LIN {X 0,Y 527.315,Z 646.786,A -85,B 0,C 180,E1 -4788.874,E2 -4788.874} C_VEL
LIN {X 0,Y 527.547,Z 631.692,A -85,B 0,C 180,E1 -4789.158,E2 -4789.158} C_VEL
LIN {X 0,Y 528.504,Z 486.386,A -85,B 0,C 180,E1 -4791.172,E2 -4791.172} C_VEL
LIN {X 0,Y 526.145,Z 470.012,A -85,B 0,C 180,E1 -4791.511,E2 -4791.511} C_VEL
LIN {X 0,Y 526.763,Z 440.59,A -85,B 0,C 180,E1 -4794.43,E2 -4794.43} C_VEL
LIN {X 0,Y 527.41,Z 413.587,A -85,B 0,C 180,E1 -4797.154,E2 -4797.154} C_VEL
LIN {X 0,Y 528.139,Z 384.774,A -85,B 0,C 180,E1 -4800.122,E2 -4800.122} C_VEL
LIN {X 0,Y 528.004,Z 381.4,A -85,B 0,C 180,E1 -4800.486,E2 -4800.486} C_VEL
LIN {X 0,Y 523.912,Z 365.853,A -85,B 0,C 180,E1 -4802.386,E2 -4802.386} C_VEL
LIN {X 0,Y 523.899,Z 365.848,A -85,B 0,C 180,E1 -4805.227,E2 -4805.227} C_VEL
LIN {X 0,Y 523.892,Z 365.854,A -85,B 0,C 180,E1 -4808.102,E2 -4808.102} C_VEL
LIN {X 0,Y 523.911,Z 365.845,A -85,B 0,C 180,E1 -4811.305,E2 -4811.305} C_VEL
LIN {X 0,Y 523.921,Z 365.841,A -85,B 0,C 180,E1 -4814.688,E2 -4814.688} C_VEL
LIN {X 0,Y 523.877,Z 365.853,A -85,B 0,C 180,E1 -4817.874,E2 -4817.874} C_VEL
LIN {X 0,Y 523.897,Z 365.845,A -85,B 0,C 180,E1 -4820.913,E2 -4820.913} C_VEL
LIN {X 0,Y 523.844,Z 365.856,A -85,B 0,C 180,E1 -4823.821,E2 -4823.821} C_VEL
LIN {X 0,Y 523.896,Z 365.851,A -85,B 0,C 180,E1 -4826.632,E2 -4826.632} C_VEL
LIN {X 0,Y 523.924,Z 365.842,A -85,B 0,C 180,E1 -4829.354,E2 -4829.354} C_VEL
LIN {X 0,Y 523.896,Z 365.854,A -85,B 0,C 180,E1 -4832.295,E2 -4832.295} C_VEL
LIN {X 0,Y 523.887,Z 365.847,A -85,B 0,C 180,E1 -4835.426,E2 -4835.426} C_VEL
LIN {X 0,Y 523.904,Z 365.85,A -85,B 0,C 180,E1 -4837.938,E2 -4837.938} C_VEL
LIN {X 0,Y 523.91,Z 365.854,A -85,B 0,C 180,E1 -4840.406,E2 -4840.406} C_VEL
LIN {X 0,Y 523.903,Z 365.849,A -85,B 0,C 180,E1 -4842.835,E2 -4842.835} C_VEL
LIN {X 0,Y 523.943,Z 365.841,A -85,B 0,C 180,E1 -4845.235,E2 -4845.235} C_VEL
LIN {X 0,Y 523.998,Z 365.842,A -85,B 0,C 180,E1 -4848.394,E2 -4848.394} C_VEL
LIN {X 0,Y 523.937,Z 365.841,A -85,B 0,C 180,E1 -4851.515,E2 -4851.515} C_VEL
LIN {X 0,Y 524.013,Z 365.84,A -85,B 0,C 180,E1 -4854.613,E2 -4854.613} C_VEL
LIN {X 0,Y 524.082,Z 365.82,A -85,B 0,C 180,E1 -4857.695,E2 -4857.695} C_VEL
LIN {X 0,Y 524.104,Z 365.825,A -85,B 0,C 180,E1 -4860.769,E2 -4860.769} C_VEL
LIN {X 0,Y 524.011,Z 365.835,A -85,B 0,C 180,E1 -4863.075,E2 -4863.075} C_VEL
LIN {X 0,Y 523.997,Z 365.832,A -85,B 0,C 180,E1 -4866.16,E2 -4866.16} C_VEL
LIN {X 0,Y 523.962,Z 365.839,A -85,B 0,C 180,E1 -4869.263,E2 -4869.263} C_VEL
LIN {X 0,Y 523.982,Z 365.835,A -85,B 0,C 180,E1 -4871.736,E2 -4871.736} C_VEL
LIN {X 0,Y 523.972,Z 365.838,A -85,B 0,C 180,E1 -4875.05,E2 -4875.05} C_VEL
LIN {X 0,Y 523.933,Z 365.842,A -85,B 0,C 180,E1 -4877.97,E2 -4877.97} C_VEL
LIN {X 0,Y 523.958,Z 365.839,A -85,B 0,C 180,E1 -4880.411,E2 -4880.411} C_VEL
LIN {X 0,Y 523.894,Z 365.854,A -85,B 0,C 180,E1 -4882.895,E2 -4882.895} C_VEL
LIN {X 0,Y 523.884,Z 365.846,A -85,B 0,C 180,E1 -4885.423,E2 -4885.423} C_VEL
LIN {X 0,Y 523.899,Z 365.844,A -85,B 0,C 180,E1 -4888.003,E2 -4888.003} C_VEL
LIN {X 0,Y 523.924,Z 365.849,A -85,B 0,C 180,E1 -4890.854,E2 -4890.854} C_VEL
LIN {X 0,Y 523.919,Z 365.845,A -85,B 0,C 180,E1 -4893.731,E2 -4893.731} C_VEL
LIN {X 0,Y 523.893,Z 365.848,A -85,B 0,C 180,E1 -4896.402,E2 -4896.402} C_VEL
LIN {X 0,Y 523.903,Z 365.852,A -85,B 0,C 180,E1 -4899.087,E2 -4899.087} C_VEL
LIN {X 0,Y 523.9,Z 365.847,A -85,B 0,C 180,E1 -4902.124,E2 -4902.124} C_VEL
LIN {X 0,Y 523.933,Z 365.847,A -85,B 0,C 180,E1 -4905.312,E2 -4905.312} C_VEL
LIN {X 0,Y 523.887,Z 365.852,A -85,B 0,C 180,E1 -4906.926,E2 -4906.926} C_VEL
LIN {X 0,Y 523.209,Z 365.936,A -85,B 0,C 180,E1 -4907.568,E2 -4907.568} C_VEL
LIN {X 0,Y 520.357,Z 366.291,A -85,B 0,C 180,E1 -4908.61,E2 -4908.61} C_VEL
LIN {X 0,Y 517.958,Z 366.589,A -85,B 0,C 180,E1 -4909.449,E2 -4909.449} C_VEL
LIN {X 0,Y 516.933,Z 366.714,A -85,B 0,C 180,E1 -4910.097,E2 -4910.097} C_VEL
LIN {X 0,Y 516.852,Z 366.724,A -85,B 0,C 180,E1 -4910.316,E2 -4910.316} C_VEL
LIN {X 0,Y 516.848,Z 366.729,A -85,B 0,C 180,E1 -4913.348,E2 -4913.348} C_VEL
LIN {X 0,Y 516.876,Z 366.723,A -85,B 0,C 180,E1 -4916.12,E2 -4916.12} C_VEL
LIN {X 0,Y 516.911,Z 366.722,A -85,B 0,C 180,E1 -4919.347,E2 -4919.347} C_VEL
LIN {X 0,Y 516.921,Z 366.886,A -85,B 0,C 180,E1 -4919.682,E2 -4919.682} C_VEL
LIN {X 0,Y 518.76,Z 371.686,A -85,B 0,C 180,E1 -4919.836,E2 -4919.836} C_VEL
LIN {X 0,Y 521.881,Z 378.811,A -85,B 0,C 180,E1 -4920.08,E2 -4920.08} C_VEL
LIN {X 0,Y 521.104,Z 494.688,A -85,B 0,C 180,E1 -4921.74,E2 -4921.74} C_VEL
LIN {X 0,Y 520.916,Z 509.79,A -85,B 0,C 180,E1 -4922.097,E2 -4922.097} C_VEL
LIN {X 0,Y 520.575,Z 523.648,A -85,B 0,C 180,E1 -4922.569,E2 -4922.569} C_VEL
LIN {X 0,Y 520.239,Z 537.825,A -85,B 0,C 180,E1 -4923.213,E2 -4923.213} C_VEL
LIN {X 0,Y 519.763,Z 550.474,A -85,B 0,C 180,E1 -4923.932,E2 -4923.932} C_VEL
LIN {X 0,Y 519.338,Z 562.529,A -85,B 0,C 180,E1 -4924.77,E2 -4924.77} C_VEL
LIN {X 0,Y 518.776,Z 574.916,A -85,B 0,C 180,E1 -4925.808,E2 -4925.808} C_VEL
LIN {X 0,Y 518.289,Z 586.545,A -85,B 0,C 180,E1 -4926.989,E2 -4926.989} C_VEL
LIN {X 0,Y 517.748,Z 597.248,A -85,B 0,C 180,E1 -4928.292,E2 -4928.292} C_VEL
LIN {X 0,Y 517.432,Z 606.116,A -85,B 0,C 180,E1 -4929.586,E2 -4929.586} C_VEL
LIN {X 0,Y 517.053,Z 614.012,A -85,B 0,C 180,E1 -4930.961,E2 -4930.961} C_VEL
LIN {X 0,Y 516.856,Z 620.282,A -85,B 0,C 180,E1 -4932.284,E2 -4932.284} C_VEL
LIN {X 0,Y 516.62,Z 626.219,A -85,B 0,C 180,E1 -4933.807,E2 -4933.807} C_VEL
LIN {X 0,Y 516.515,Z 631.091,A -85,B 0,C 180,E1 -4935.421,E2 -4935.421} C_VEL
LIN {X 0,Y 516.398,Z 633.9,A -85,B 0,C 180,E1 -4936.623,E2 -4936.623} C_VEL
LIN {X 0,Y 516.377,Z 636.848,A -85,B 0,C 180,E1 -4938.504,E2 -4938.504} C_VEL
LIN {X 0,Y 516.313,Z 637.923,A -85,B 0,C 180,E1 -4939.808,E2 -4939.808} C_VEL
LIN {X 0,Y 516.336,Z 638.23,A -85,B 0,C 180,E1 -4941.39,E2 -4941.39} C_VEL
LIN {X 0,Y 516.401,Z 637.436,A -85,B 0,C 180,E1 -4942.965,E2 -4942.965} C_VEL
LIN {X 0,Y 516.42,Z 635.551,A -85,B 0,C 180,E1 -4944.534,E2 -4944.534} C_VEL
LIN {X 0,Y 516.458,Z 632.481,A -85,B 0,C 180,E1 -4946.099,E2 -4946.099} C_VEL
LIN {X 0,Y 516.538,Z 628.218,A -85,B 0,C 180,E1 -4947.661,E2 -4947.661} C_VEL
LIN {X 0,Y 516.697,Z 622.669,A -85,B 0,C 180,E1 -4949.221,E2 -4949.221} C_VEL
LIN {X 0,Y 517.013,Z 615.669,A -85,B 0,C 180,E1 -4950.779,E2 -4950.779} C_VEL
LIN {X 0,Y 517.298,Z 608.205,A -85,B 0,C 180,E1 -4952.141,E2 -4952.141} C_VEL
LIN {X 0,Y 517.678,Z 599.262,A -85,B 0,C 180,E1 -4953.503,E2 -4953.503} C_VEL
LIN {X 0,Y 518.198,Z 588.478,A -85,B 0,C 180,E1 -4954.863,E2 -4954.863} C_VEL
LIN {X 0,Y 518.651,Z 577.402,A -85,B 0,C 180,E1 -4956.028,E2 -4956.028} C_VEL
LIN {X 0,Y 519.169,Z 565.212,A -85,B 0,C 180,E1 -4957.096,E2 -4957.096} C_VEL
LIN {X 0,Y 519.659,Z 553.226,A -85,B 0,C 180,E1 -4957.968,E2 -4957.968} C_VEL
LIN {X 0,Y 520.137,Z 539.655,A -85,B 0,C 180,E1 -4958.775,E2 -4958.775} C_VEL
LIN {X 0,Y 520.55,Z 526.025,A -85,B 0,C 180,E1 -4959.418,E2 -4959.418} C_VEL
LIN {X 0,Y 520.835,Z 510.868,A -85,B 0,C 180,E1 -4959.958,E2 -4959.958} C_VEL
LIN {X 0,Y 521.031,Z 496.258,A -85,B 0,C 180,E1 -4960.32,E2 -4960.32} C_VEL
LIN {X 0,Y 521.839,Z 378.575,A -85,B 0,C 180,E1 -4962.012,E2 -4962.012} C_VEL
LIN {X 0,Y 517.046,Z 367.428,A -85,B 0,C 180,E1 -4962.39,E2 -4962.39} C_VEL
LIN {X 0,Y 516.912,Z 366.723,A -85,B 0,C 180,E1 -4962.424,E2 -4962.424} C_VEL
LIN {X 0,Y 516.833,Z 366.728,A -85,B 0,C 180,E1 -4965.781,E2 -4965.781} C_VEL
LIN {X 0,Y 516.872,Z 366.722,A -85,B 0,C 180,E1 -4968.224,E2 -4968.224} C_VEL
LIN {X 0,Y 516.879,Z 366.726,A -85,B 0,C 180,E1 -4970.703,E2 -4970.703} C_VEL
LIN {X 0,Y 516.836,Z 366.733,A -85,B 0,C 180,E1 -4973.225,E2 -4973.225} C_VEL
LIN {X 0,Y 516.858,Z 366.724,A -85,B 0,C 180,E1 -4976.176,E2 -4976.176} C_VEL
LIN {X 0,Y 516.828,Z 366.729,A -85,B 0,C 180,E1 -4978.42,E2 -4978.42} C_VEL
LIN {X 0,Y 516.847,Z 366.729,A -85,B 0,C 180,E1 -4981.112,E2 -4981.112} C_VEL
LIN {X 0,Y 516.867,Z 366.721,A -85,B 0,C 180,E1 -4983.959,E2 -4983.959} C_VEL
LIN {X 0,Y 516.806,Z 366.733,A -85,B 0,C 180,E1 -4986.751,E2 -4986.751} C_VEL
LIN {X 0,Y 516.841,Z 366.725,A -85,B 0,C 180,E1 -4989.724,E2 -4989.724} C_VEL
LIN {X 0,Y 516.833,Z 366.73,A -85,B 0,C 180,E1 -4992.836,E2 -4992.836} C_VEL
LIN {X 0,Y 516.892,Z 366.724,A -85,B 0,C 180,E1 -4995.006,E2 -4995.006} C_VEL
LIN {X 0,Y 516.844,Z 366.724,A -85,B 0,C 180,E1 -4998.406,E2 -4998.406} C_VEL
LIN {X 0,Y 516.855,Z 366.73,A -85,B 0,C 180,E1 -5001.281,E2 -5001.281} C_VEL
LIN {X 0,Y 516.846,Z 366.725,A -85,B 0,C 180,E1 -5004.217,E2 -5004.217} C_VEL
LIN {X 0,Y 516.852,Z 366.727,A -85,B 0,C 180,E1 -5007.05,E2 -5007.05} C_VEL
LIN {X 0,Y 516.83,Z 366.728,A -85,B 0,C 180,E1 -5009.792,E2 -5009.792} C_VEL
LIN {X 0,Y 516.858,Z 366.723,A -85,B 0,C 180,E1 -5012.463,E2 -5012.463} C_VEL
LIN {X 0,Y 516.847,Z 366.727,A -85,B 0,C 180,E1 -5015.649,E2 -5015.649} C_VEL
LIN {X 0,Y 516.874,Z 366.721,A -85,B 0,C 180,E1 -5018.461,E2 -5018.461} C_VEL
LIN {X 0,Y 516.873,Z 366.722,A -85,B 0,C 180,E1 -5020.953,E2 -5020.953} C_VEL
LIN {X 0,Y 516.874,Z 366.73,A -85,B 0,C 180,E1 -5023.409,E2 -5023.409} C_VEL
LIN {X 0,Y 516.863,Z 366.722,A -85,B 0,C 180,E1 -5025.832,E2 -5025.832} C_VEL
LIN {X 0,Y 516.929,Z 366.705,A -85,B 0,C 180,E1 -5029.027,E2 -5029.027} C_VEL
LIN {X 0,Y 516.91,Z 366.714,A -85,B 0,C 180,E1 -5032.186,E2 -5032.186} C_VEL
LIN {X 0,Y 516.973,Z 366.708,A -85,B 0,C 180,E1 -5034.539,E2 -5034.539} C_VEL
LIN {X 0,Y 517.056,Z 366.701,A -85,B 0,C 180,E1 -5037.663,E2 -5037.663} C_VEL
LIN {X 0,Y 517.045,Z 366.702,A -85,B 0,C 180,E1 -5040,E2 -5040} C_VEL
LIN {X 0,Y 517.058,Z 366.697,A -85,B 0,C 180,E1 -5042.337,E2 -5042.337} C_VEL
LIN {X 0,Y 516.965,Z 366.714,A -85,B 0,C 180,E1 -5045.461,E2 -5045.461} C_VEL
LIN {X 0,Y 516.911,Z 366.714,A -85,B 0,C 180,E1 -5048.601,E2 -5048.601} C_VEL
LIN {X 0,Y 516.942,Z 366.719,A -85,B 0,C 180,E1 -5051.807,E2 -5051.807} C_VEL
LIN {X 0,Y 516.924,Z 366.714,A -85,B 0,C 180,E1 -5055.142,E2 -5055.142} C_VEL
LIN {X 0,Y 516.858,Z 366.723,A -85,B 0,C 180,E1 -5058.224,E2 -5058.224} C_VEL
LIN {X 0,Y 516.86,Z 366.723,A -85,B 0,C 180,E1 -5060.703,E2 -5060.703} C_VEL
LIN {X 0,Y 516.831,Z 366.727,A -85,B 0,C 180,E1 -5063.225,E2 -5063.225} C_VEL
LIN {X 0,Y 516.869,Z 366.723,A -85,B 0,C 180,E1 -5066.182,E2 -5066.182} C_VEL
LIN {X 0,Y 516.875,Z 366.727,A -85,B 0,C 180,E1 -5069.519,E2 -5069.519} C_VEL
LIN {X 0,Y 516.858,Z 366.722,A -85,B 0,C 180,E1 -5072.538,E2 -5072.538} C_VEL
LIN {X 0,Y 516.841,Z 366.727,A -85,B 0,C 180,E1 -5075.327,E2 -5075.327} C_VEL
LIN {X 0,Y 516.854,Z 366.72,A -85,B 0,C 180,E1 -5078.718,E2 -5078.718} C_VEL
LIN {X 0,Y 516.835,Z 366.732,A -85,B 0,C 180,E1 -5081.783,E2 -5081.783} C_VEL
LIN {X 0,Y 516.89,Z 366.719,A -85,B 0,C 180,E1 -5085.007,E2 -5085.007} C_VEL
LIN {X 0,Y 516.829,Z 366.726,A -85,B 0,C 180,E1 -5088.218,E2 -5088.218} C_VEL
LIN {X 0,Y 516.863,Z 366.725,A -85,B 0,C 180,E1 -5091.283,E2 -5091.283} C_VEL
LIN {X 0,Y 516.845,Z 366.728,A -85,B 0,C 180,E1 -5094.674,E2 -5094.674} C_VEL
LIN {X 0,Y 516.918,Z 366.823,A -85,B 0,C 180,E1 -5097.351,E2 -5097.351} C_VEL
LIN {X 0,Y 521.433,Z 384.33,A -85,B 0,C 180,E1 -5099.474,E2 -5099.474} C_VEL
LIN {X 0,Y 520.757,Z 408.762,A -85,B 0,C 180,E1 -5102.033,E2 -5102.033} C_VEL
LIN {X 0,Y 520.055,Z 436.422,A -85,B 0,C 180,E1 -5104.882,E2 -5104.882} C_VEL
LIN {X 0,Y 519.34,Z 465.735,A -85,B 0,C 180,E1 -5107.849,E2 -5107.849} C_VEL
LIN {X 0,Y 519.219,Z 469.127,A -85,B 0,C 180,E1 -5108.189,E2 -5108.189} C_VEL
LIN {X 0,Y 521.848,Z 486.32,A -85,B 0,C 180,E1 -5108.556,E2 -5108.556} C_VEL
LIN {X 0,Y 520.76,Z 638.646,A -85,B 0,C 180,E1 -5110.718,E2 -5110.718} C_VEL
LIN {X 0,Y 520.393,Z 654.328,A -85,B 0,C 180,E1 -5111.102,E2 -5111.102} C_VEL
LIN {X 0,Y 519.991,Z 669.425,A -85,B 0,C 180,E1 -5111.634,E2 -5111.634} C_VEL
LIN {X 0,Y 519.522,Z 683.387,A -85,B 0,C 180,E1 -5112.28,E2 -5112.28} C_VEL
LIN {X 0,Y 519.026,Z 697.119,A -85,B 0,C 180,E1 -5113.075,E2 -5113.075} C_VEL
LIN {X 0,Y 518.522,Z 711.14,A -85,B 0,C 180,E1 -5114.07,E2 -5114.07} C_VEL
LIN {X 0,Y 517.987,Z 723.857,A -85,B 0,C 180,E1 -5115.162,E2 -5115.162} C_VEL
LIN {X 0,Y 517.538,Z 736.378,A -85,B 0,C 180,E1 -5116.453,E2 -5116.453} C_VEL
LIN {X 0,Y 517.111,Z 747.534,A -85,B 0,C 180,E1 -5117.839,E2 -5117.839} C_VEL
LIN {X 0,Y 516.895,Z 756.856,A -85,B 0,C 180,E1 -5119.225,E2 -5119.225} C_VEL
LIN {X 0,Y 516.611,Z 764.583,A -85,B 0,C 180,E1 -5120.604,E2 -5120.604} C_VEL
LIN {X 0,Y 516.508,Z 770.059,A -85,B 0,C 180,E1 -5121.786,E2 -5121.786} C_VEL
LIN {X 0,Y 516.391,Z 774.605,A -85,B 0,C 180,E1 -5122.964,E2 -5122.964} C_VEL
LIN {X 0,Y 516.373,Z 779.385,A -85,B 0,C 180,E1 -5124.533,E2 -5124.533} C_VEL
LIN {X 0,Y 516.307,Z 782.886,A -85,B 0,C 180,E1 -5126.097,E2 -5126.097} C_VEL
LIN {X 0,Y 516.257,Z 785.188,A -85,B 0,C 180,E1 -5127.659,E2 -5127.659} C_VEL
LIN {X 0,Y 516.157,Z 786.347,A -85,B 0,C 180,E1 -5129.22,E2 -5129.22} C_VEL
LIN {X 0,Y 516.157,Z 786.346,A -85,B 0,C 180,E1 -5130.78,E2 -5130.78} C_VEL
LIN {X 0,Y 516.257,Z 785.185,A -85,B 0,C 180,E1 -5132.34,E2 -5132.34} C_VEL
LIN {X 0,Y 516.307,Z 782.882,A -85,B 0,C 180,E1 -5133.902,E2 -5133.902} C_VEL
LIN {X 0,Y 516.372,Z 779.387,A -85,B 0,C 180,E1 -5135.467,E2 -5135.467} C_VEL
LIN {X 0,Y 516.391,Z 774.611,A -85,B 0,C 180,E1 -5137.035,E2 -5137.035} C_VEL
LIN {X 0,Y 516.54,Z 768.361,A -85,B 0,C 180,E1 -5138.607,E2 -5138.607} C_VEL
LIN {X 0,Y 516.676,Z 761.44,A -85,B 0,C 180,E1 -5139.987,E2 -5139.987} C_VEL
LIN {X 0,Y 516.952,Z 753.027,A -85,B 0,C 180,E1 -5141.368,E2 -5141.368} C_VEL
LIN {X 0,Y 517.283,Z 742.958,A -85,B 0,C 180,E1 -5142.754,E2 -5142.754} C_VEL
LIN {X 0,Y 517.649,Z 732.687,A -85,B 0,C 180,E1 -5143.944,E2 -5143.944} C_VEL
LIN {X 0,Y 518.079,Z 720.663,A -85,B 0,C 180,E1 -5145.124,E2 -5145.124} C_VEL
LIN {X 0,Y 518.59,Z 708.438,A -85,B 0,C 180,E1 -5146.129,E2 -5146.129} C_VEL
LIN {X 0,Y 519.071,Z 695.419,A -85,B 0,C 180,E1 -5147.024,E2 -5147.024} C_VEL
LIN {X 0,Y 519.566,Z 681.262,A -85,B 0,C 180,E1 -5147.82,E2 -5147.82} C_VEL
LIN {X 0,Y 520.026,Z 666.743,A -85,B 0,C 180,E1 -5148.466,E2 -5148.466} C_VEL
LIN {X 0,Y 520.439,Z 651.075,A -85,B 0,C 180,E1 -5148.986,E2 -5148.986} C_VEL
LIN {X 0,Y 520.798,Z 636.224,A -85,B 0,C 180,E1 -5149.321,E2 -5149.321} C_VEL
LIN {X 0,Y 521.835,Z 486.88,A -85,B 0,C 180,E1 -5151.433,E2 -5151.433} C_VEL
LIN {X 0,Y 519.194,Z 468.922,A -85,B 0,C 180,E1 -5151.812,E2 -5151.812} C_VEL
LIN {X 0,Y 519.864,Z 440.568,A -85,B 0,C 180,E1 -5154.669,E2 -5154.669} C_VEL
LIN {X 0,Y 520.564,Z 414.648,A -85,B 0,C 180,E1 -5157.323,E2 -5157.323} C_VEL
LIN {X 0,Y 521.371,Z 386.766,A -85,B 0,C 180,E1 -5160.24,E2 -5160.24} C_VEL
LIN {X 0,Y 521.416,Z 384.129,A -85,B 0,C 180,E1 -5160.522,E2 -5160.522} C_VEL
LIN {X 0,Y 516.889,Z 366.725,A -85,B 0,C 180,E1 -5162.708,E2 -5162.708} C_VEL
LIN {X 0,Y 516.807,Z 366.734,A -85,B 0,C 180,E1 -5165.784,E2 -5165.784} C_VEL
LIN {X 0,Y 516.864,Z 366.726,A -85,B 0,C 180,E1 -5168.716,E2 -5168.716} C_VEL
LIN {X 0,Y 516.872,Z 366.725,A -85,B 0,C 180,E1 -5171.777,E2 -5171.777} C_VEL
LIN {X 0,Y 516.886,Z 366.715,A -85,B 0,C 180,E1 -5175.006,E2 -5175.006} C_VEL
LIN {X 0,Y 516.838,Z 366.73,A -85,B 0,C 180,E1 -5178.406,E2 -5178.406} C_VEL
LIN {X 0,Y 516.859,Z 366.721,A -85,B 0,C 180,E1 -5181.282,E2 -5181.282} C_VEL
LIN {X 0,Y 516.837,Z 366.73,A -85,B 0,C 180,E1 -5184.672,E2 -5184.672} C_VEL
LIN {X 0,Y 516.854,Z 366.724,A -85,B 0,C 180,E1 -5187.461,E2 -5187.461} C_VEL
LIN {X 0,Y 516.871,Z 366.73,A -85,B 0,C 180,E1 -5190.481,E2 -5190.481} C_VEL
LIN {X 0,Y 516.864,Z 366.725,A -85,B 0,C 180,E1 -5193.818,E2 -5193.818} C_VEL
LIN {X 0,Y 516.826,Z 366.732,A -85,B 0,C 180,E1 -5196.775,E2 -5196.775} C_VEL
LIN {X 0,Y 516.86,Z 366.723,A -85,B 0,C 180,E1 -5199.751,E2 -5199.751} C_VEL
LIN {X 0,Y 516.862,Z 366.729,A -85,B 0,C 180,E1 -5202.594,E2 -5202.594} C_VEL
LIN {X 0,Y 516.914,Z 366.718,A -85,B 0,C 180,E1 -5205.029,E2 -5205.029} C_VEL
LIN {X 0,Y 516.951,Z 366.718,A -85,B 0,C 180,E1 -5208.234,E2 -5208.234} C_VEL
LIN {X 0,Y 516.909,Z 366.717,A -85,B 0,C 180,E1 -5211.399,E2 -5211.399} C_VEL
LIN {X 0,Y 516.963,Z 366.717,A -85,B 0,C 180,E1 -5214.539,E2 -5214.539} C_VEL
LIN {X 0,Y 517.054,Z 366.696,A -85,B 0,C 180,E1 -5217.663,E2 -5217.663} C_VEL
LIN {X 0,Y 517.074,Z 366.7,A -85,B 0,C 180,E1 -5220.779,E2 -5220.779} C_VEL
LIN {X 0,Y 516.953,Z 366.714,A -85,B 0,C 180,E1 -5223.118,E2 -5223.118} C_VEL
LIN {X 0,Y 516.966,Z 366.708,A -85,B 0,C 180,E1 -5226.244,E2 -5226.244} C_VEL
LIN {X 0,Y 516.918,Z 366.715,A -85,B 0,C 180,E1 -5229.39,E2 -5229.39} C_VEL
LIN {X 0,Y 516.938,Z 366.713,A -85,B 0,C 180,E1 -5231.807,E2 -5231.807} C_VEL
LIN {X 0,Y 516.924,Z 366.714,A -85,B 0,C 180,E1 -5235.144,E2 -5235.144} C_VEL
LIN {X 0,Y 516.901,Z 366.72,A -85,B 0,C 180,E1 -5238.223,E2 -5238.223} C_VEL
LIN {X 0,Y 516.898,Z 366.717,A -85,B 0,C 180,E1 -5240.702,E2 -5240.702} C_VEL
LIN {X 0,Y 516.871,Z 366.723,A -85,B 0,C 180,E1 -5244.074,E2 -5244.074} C_VEL
LIN {X 0,Y 516.827,Z 366.728,A -85,B 0,C 180,E1 -5246.664,E2 -5246.664} C_VEL
LIN {X 0,Y 516.895,Z 366.721,A -85,B 0,C 180,E1 -5249.524,E2 -5249.524} C_VEL
LIN {X 0,Y 516.883,Z 366.719,A -85,B 0,C 180,E1 -5252.544,E2 -5252.544} C_VEL
LIN {X 0,Y 516.855,Z 366.726,A -85,B 0,C 180,E1 -5255.33,E2 -5255.33} C_VEL
LIN {X 0,Y 516.869,Z 366.722,A -85,B 0,C 180,E1 -5257.944,E2 -5257.944} C_VEL
LIN {X 0,Y 516.845,Z 366.728,A -85,B 0,C 180,E1 -5260.746,E2 -5260.746} C_VEL
LIN {X 0,Y 516.873,Z 366.718,A -85,B 0,C 180,E1 -5263.905,E2 -5263.905} C_VEL
LIN {X 0,Y 516.837,Z 366.728,A -85,B 0,C 180,E1 -5266.928,E2 -5266.928} C_VEL
LIN {X 0,Y 516.854,Z 366.725,A -85,B 0,C 180,E1 -5269.594,E2 -5269.594} C_VEL
LIN {X 0,Y 516.852,Z 366.724,A -85,B 0,C 180,E1 -5270.316,E2 -5270.316} C_VEL
LIN {X 0,Y 516.193,Z 366.814,A -85,B 0,C 180,E1 -5270.966,E2 -5270.966} C_VEL
LIN {X 0,Y 513.344,Z 367.167,A -85,B 0,C 180,E1 -5272.022,E2 -5272.022} C_VEL
LIN {X 0,Y 510.929,Z 367.467,A -85,B 0,C 180,E1 -5272.873,E2 -5272.873} C_VEL
LIN {X 0,Y 509.887,Z 367.594,A -85,B 0,C 180,E1 -5273.529,E2 -5273.529} C_VEL
LIN {X 0,Y 509.8,Z 367.603,A -85,B 0,C 180,E1 -5273.752,E2 -5273.752} C_VEL
LIN {X 0,Y 509.835,Z 367.603,A -85,B 0,C 180,E1 -5276.539,E2 -5276.539} C_VEL
LIN {X 0,Y 509.877,Z 367.625,A -85,B 0,C 180,E1 -5279.363,E2 -5279.363} C_VEL
LIN {X 0,Y 511.415,Z 371.854,A -85,B 0,C 180,E1 -5279.499,E2 -5279.499} C_VEL
LIN {X 0,Y 515.302,Z 380.765,A -85,B 0,C 180,E1 -5279.812,E2 -5279.812} C_VEL
LIN {X 0,Y 514.445,Z 495.575,A -85,B 0,C 180,E1 -5281.479,E2 -5281.479} C_VEL
LIN {X 0,Y 514.256,Z 510.81,A -85,B 0,C 180,E1 -5281.842,E2 -5281.842} C_VEL
LIN {X 0,Y 513.941,Z 525.052,A -85,B 0,C 180,E1 -5282.337,E2 -5282.337} C_VEL
LIN {X 0,Y 513.586,Z 538.387,A -85,B 0,C 180,E1 -5282.95,E2 -5282.95} C_VEL
LIN {X 0,Y 513.075,Z 551.1,A -85,B 0,C 180,E1 -5283.676,E2 -5283.676} C_VEL
LIN {X 0,Y 512.635,Z 563.228,A -85,B 0,C 180,E1 -5284.525,E2 -5284.525} C_VEL
LIN {X 0,Y 512.015,Z 575.76,A -85,B 0,C 180,E1 -5285.584,E2 -5285.584} C_VEL
LIN {X 0,Y 511.529,Z 586.663,A -85,B 0,C 180,E1 -5286.693,E2 -5286.693} C_VEL
LIN {X 0,Y 510.957,Z 597.337,A -85,B 0,C 180,E1 -5287.988,E2 -5287.988} C_VEL
LIN {X 0,Y 510.57,Z 606.929,A -85,B 0,C 180,E1 -5289.394,E2 -5289.394} C_VEL
LIN {X 0,Y 510.127,Z 615.442,A -85,B 0,C 180,E1 -5290.902,E2 -5290.902} C_VEL
LIN {X 0,Y 509.858,Z 622.115,A -85,B 0,C 180,E1 -5292.348,E2 -5292.348} C_VEL
LIN {X 0,Y 509.648,Z 628.21,A -85,B 0,C 180,E1 -5293.991,E2 -5293.991} C_VEL
LIN {X 0,Y 509.479,Z 632.835,A -85,B 0,C 180,E1 -5295.624,E2 -5295.624} C_VEL
LIN {X 0,Y 509.353,Z 636.146,A -85,B 0,C 180,E1 -5297.247,E2 -5297.247} C_VEL
LIN {X 0,Y 509.362,Z 638.239,A -85,B 0,C 180,E1 -5298.863,E2 -5298.863} C_VEL
LIN {X 0,Y 509.302,Z 639.205,A -85,B 0,C 180,E1 -5300.469,E2 -5300.469} C_VEL
LIN {X 0,Y 509.337,Z 639.056,A -85,B 0,C 180,E1 -5302.069,E2 -5302.069} C_VEL
LIN {X 0,Y 509.416,Z 637.793,A -85,B 0,C 180,E1 -5303.664,E2 -5303.664} C_VEL
LIN {X 0,Y 509.388,Z 635.392,A -85,B 0,C 180,E1 -5305.252,E2 -5305.252} C_VEL
LIN {X 0,Y 509.576,Z 631.807,A -85,B 0,C 180,E1 -5306.838,E2 -5306.838} C_VEL
LIN {X 0,Y 509.593,Z 627.042,A -85,B 0,C 180,E1 -5308.42,E2 -5308.42} C_VEL
LIN {X 0,Y 509.854,Z 620.902,A -85,B 0,C 180,E1 -5310,E2 -5310} C_VEL
LIN {X 0,Y 510.217,Z 613.234,A -85,B 0,C 180,E1 -5311.579,E2 -5311.579} C_VEL
LIN {X 0,Y 510.565,Z 605.095,A -85,B 0,C 180,E1 -5312.959,E2 -5312.959} C_VEL
LIN {X 0,Y 511.094,Z 595.303,A -85,B 0,C 180,E1 -5314.338,E2 -5314.338} C_VEL
LIN {X 0,Y 511.572,Z 585.332,A -85,B 0,C 180,E1 -5315.519,E2 -5315.519} C_VEL
LIN {X 0,Y 512.067,Z 573.425,A -85,B 0,C 180,E1 -5316.7,E2 -5316.7} C_VEL
LIN {X 0,Y 512.638,Z 561.493,A -85,B 0,C 180,E1 -5317.682,E2 -5317.682} C_VEL
LIN {X 0,Y 513.193,Z 548.475,A -85,B 0,C 180,E1 -5318.565,E2 -5318.565} C_VEL
LIN {X 0,Y 513.613,Z 535.982,A -85,B 0,C 180,E1 -5319.252,E2 -5319.252} C_VEL
LIN {X 0,Y 514.013,Z 522.246,A -85,B 0,C 180,E1 -5319.851,E2 -5319.851} C_VEL
LIN {X 0,Y 514.252,Z 507.515,A -85,B 0,C 180,E1 -5320.333,E2 -5320.333} C_VEL
LIN {X 0,Y 514.401,Z 492.958,A -85,B 0,C 180,E1 -5320.654,E2 -5320.654} C_VEL
LIN {X 0,Y 515.255,Z 380.378,A -85,B 0,C 180,E1 -5322.28,E2 -5322.28} C_VEL
LIN {X 0,Y 509.971,Z 368.313,A -85,B 0,C 180,E1 -5322.703,E2 -5322.703} C_VEL
LIN {X 0,Y 509.851,Z 367.604,A -85,B 0,C 180,E1 -5322.741,E2 -5322.741} C_VEL
LIN {X 0,Y 509.801,Z 367.604,A -85,B 0,C 180,E1 -5326.005,E2 -5326.005} C_VEL
LIN {X 0,Y 509.829,Z 367.602,A -85,B 0,C 180,E1 -5328.485,E2 -5328.485} C_VEL
LIN {X 0,Y 509.824,Z 367.608,A -85,B 0,C 180,E1 -5331.003,E2 -5331.003} C_VEL
LIN {X 0,Y 509.797,Z 367.606,A -85,B 0,C 180,E1 -5333.565,E2 -5333.565} C_VEL
LIN {X 0,Y 509.799,Z 367.605,A -85,B 0,C 180,E1 -5336.352,E2 -5336.352} C_VEL
LIN {X 0,Y 509.792,Z 367.611,A -85,B 0,C 180,E1 -5338.849,E2 -5338.849} C_VEL
LIN {X 0,Y 509.786,Z 367.607,A -85,B 0,C 180,E1 -5341.592,E2 -5341.592} C_VEL
LIN {X 0,Y 509.826,Z 367.599,A -85,B 0,C 180,E1 -5344.415,E2 -5344.415} C_VEL
LIN {X 0,Y 509.774,Z 367.612,A -85,B 0,C 180,E1 -5347.344,E2 -5347.344} C_VEL
LIN {X 0,Y 509.79,Z 367.602,A -85,B 0,C 180,E1 -5350.386,E2 -5350.386} C_VEL
LIN {X 0,Y 509.787,Z 367.606,A -85,B 0,C 180,E1 -5353.574,E2 -5353.574} C_VEL
LIN {X 0,Y 509.787,Z 367.604,A -85,B 0,C 180,E1 -5356.424,E2 -5356.424} C_VEL
LIN {X 0,Y 509.807,Z 367.605,A -85,B 0,C 180,E1 -5359.614,E2 -5359.614} C_VEL
LIN {X 0,Y 509.781,Z 367.605,A -85,B 0,C 180,E1 -5362.656,E2 -5362.656} C_VEL
LIN {X 0,Y 509.825,Z 367.598,A -85,B 0,C 180,E1 -5365.801,E2 -5365.801} C_VEL
LIN {X 0,Y 509.807,Z 367.604,A -85,B 0,C 180,E1 -5368.726,E2 -5368.726} C_VEL
LIN {X 0,Y 509.815,Z 367.601,A -85,B 0,C 180,E1 -5372.05,E2 -5372.05} C_VEL
LIN {X 0,Y 509.773,Z 367.607,A -85,B 0,C 180,E1 -5374.698,E2 -5374.698} C_VEL
LIN {X 0,Y 509.816,Z 367.608,A -85,B 0,C 180,E1 -5377.458,E2 -5377.458} C_VEL
LIN {X 0,Y 509.898,Z 367.591,A -85,B 0,C 180,E1 -5379.844,E2 -5379.844} C_VEL
LIN {X 0,Y 509.843,Z 367.601,A -85,B 0,C 180,E1 -5383.173,E2 -5383.173} C_VEL
LIN {X 0,Y 509.836,Z 367.6,A -85,B 0,C 180,E1 -5385.633,E2 -5385.633} C_VEL
LIN {X 0,Y 509.894,Z 367.579,A -85,B 0,C 180,E1 -5388.874,E2 -5388.874} C_VEL
LIN {X 0,Y 509.863,Z 367.593,A -85,B 0,C 180,E1 -5392.077,E2 -5392.077} C_VEL
LIN {X 0,Y 509.928,Z 367.586,A -85,B 0,C 180,E1 -5394.463,E2 -5394.463} C_VEL
LIN {X 0,Y 510.025,Z 367.577,A -85,B 0,C 180,E1 -5397.631,E2 -5397.631} C_VEL
LIN {X 0,Y 510.015,Z 367.578,A -85,B 0,C 180,E1 -5400,E2 -5400} C_VEL
LIN {X 0,Y 510.029,Z 367.572,A -85,B 0,C 180,E1 -5402.369,E2 -5402.369} C_VEL
LIN {X 0,Y 509.918,Z 367.593,A -85,B 0,C 180,E1 -5405.536,E2 -5405.536} C_VEL
LIN {X 0,Y 509.865,Z 367.596,A -85,B 0,C 180,E1 -5407.923,E2 -5407.923} C_VEL
LIN {X 0,Y 509.896,Z 367.592,A -85,B 0,C 180,E1 -5411.126,E2 -5411.126} C_VEL
LIN {X 0,Y 509.83,Z 367.596,A -85,B 0,C 180,E1 -5414.367,E2 -5414.367} C_VEL
LIN {X 0,Y 509.778,Z 367.606,A -85,B 0,C 180,E1 -5416.829,E2 -5416.829} C_VEL
LIN {X 0,Y 509.814,Z 367.602,A -85,B 0,C 180,E1 -5419.32,E2 -5419.32} C_VEL
LIN {X 0,Y 509.814,Z 367.599,A -85,B 0,C 180,E1 -5422.541,E2 -5422.541} C_VEL
LIN {X 0,Y 509.791,Z 367.607,A -85,B 0,C 180,E1 -5425.3,E2 -5425.3} C_VEL
LIN {X 0,Y 509.8,Z 367.606,A -85,B 0,C 180,E1 -5428.082,E2 -5428.082} C_VEL
LIN {X 0,Y 509.819,Z 367.601,A -85,B 0,C 180,E1 -5430.667,E2 -5430.667} C_VEL
LIN {X 0,Y 509.824,Z 367.602,A -85,B 0,C 180,E1 -5433.463,E2 -5433.463} C_VEL
LIN {X 0,Y 509.757,Z 367.611,A -85,B 0,C 180,E1 -5436.359,E2 -5436.359} C_VEL
LIN {X 0,Y 509.802,Z 367.603,A -85,B 0,C 180,E1 -5439.467,E2 -5439.467} C_VEL
LIN {X 0,Y 509.778,Z 367.605,A -85,B 0,C 180,E1 -5442.495,E2 -5442.495} C_VEL
LIN {X 0,Y 509.833,Z 367.6,A -85,B 0,C 180,E1 -5445.33,E2 -5445.33} C_VEL
LIN {X 0,Y 509.78,Z 367.601,A -85,B 0,C 180,E1 -5448.568,E2 -5448.568} C_VEL
LIN {X 0,Y 509.808,Z 367.608,A -85,B 0,C 180,E1 -5451.659,E2 -5451.659} C_VEL
LIN {X 0,Y 509.803,Z 367.606,A -85,B 0,C 180,E1 -5454.62,E2 -5454.62} C_VEL
LIN {X 0,Y 509.858,Z 367.616,A -85,B 0,C 180,E1 -5457.063,E2 -5457.063} C_VEL
LIN {X 0,Y 514.667,Z 386.214,A -85,B 0,C 180,E1 -5459.349,E2 -5459.349} C_VEL
LIN {X 0,Y 513.946,Z 409.84,A -85,B 0,C 180,E1 -5461.851,E2 -5461.851} C_VEL
LIN {X 0,Y 513.192,Z 436.826,A -85,B 0,C 180,E1 -5464.668,E2 -5464.668} C_VEL
LIN {X 0,Y 512.373,Z 466.644,A -85,B 0,C 180,E1 -5467.734,E2 -5467.734} C_VEL
LIN {X 0,Y 512.308,Z 468.297,A -85,B 0,C 180,E1 -5467.892,E2 -5467.892} C_VEL
LIN {X 0,Y 515.198,Z 487.539,A -85,B 0,C 180,E1 -5468.298,E2 -5468.298} C_VEL
LIN {X 0,Y 514.052,Z 636.943,A -85,B 0,C 180,E1 -5470.443,E2 -5470.443} C_VEL
LIN {X 0,Y 513.616,Z 652.848,A -85,B 0,C 180,E1 -5470.828,E2 -5470.828} C_VEL
LIN {X 0,Y 513.169,Z 668.596,A -85,B 0,C 180,E1 -5471.39,E2 -5471.39} C_VEL
LIN {X 0,Y 512.638,Z 682.352,A -85,B 0,C 180,E1 -5472.034,E2 -5472.034} C_VEL
LIN {X 0,Y 512.142,Z 696.091,A -85,B 0,C 180,E1 -5472.84,E2 -5472.84} C_VEL
LIN {X 0,Y 511.608,Z 708.787,A -85,B 0,C 180,E1 -5473.746,E2 -5473.746} C_VEL
LIN {X 0,Y 511.006,Z 721.725,A -85,B 0,C 180,E1 -5474.852,E2 -5474.852} C_VEL
LIN {X 0,Y 510.564,Z 733.526,A -85,B 0,C 180,E1 -5476.061,E2 -5476.061} C_VEL
LIN {X 0,Y 510.191,Z 743.484,A -85,B 0,C 180,E1 -5477.267,E2 -5477.267} C_VEL
LIN {X 0,Y 509.889,Z 753.423,A -85,B 0,C 180,E1 -5478.693,E2 -5478.693} C_VEL
LIN {X 0,Y 509.576,Z 761.468,A -85,B 0,C 180,E1 -5480.073,E2 -5480.073} C_VEL
LIN {X 0,Y 509.431,Z 769.133,A -85,B 0,C 180,E1 -5481.671,E2 -5481.671} C_VEL
LIN {X 0,Y 509.289,Z 775.219,A -85,B 0,C 180,E1 -5483.264,E2 -5483.264} C_VEL
LIN {X 0,Y 509.305,Z 778.85,A -85,B 0,C 180,E1 -5484.457,E2 -5484.457} C_VEL
LIN {X 0,Y 509.217,Z 782.511,A -85,B 0,C 180,E1 -5486.043,E2 -5486.043} C_VEL
LIN {X 0,Y 509.185,Z 784.924,A -85,B 0,C 180,E1 -5487.627,E2 -5487.627} C_VEL
LIN {X 0,Y 509.071,Z 786.123,A -85,B 0,C 180,E1 -5489.209,E2 -5489.209} C_VEL
LIN {X 0,Y 509.071,Z 786.122,A -85,B 0,C 180,E1 -5490.791,E2 -5490.791} C_VEL
LIN {X 0,Y 509.185,Z 784.921,A -85,B 0,C 180,E1 -5492.373,E2 -5492.373} C_VEL
LIN {X 0,Y 509.217,Z 782.506,A -85,B 0,C 180,E1 -5493.957,E2 -5493.957} C_VEL
LIN {X 0,Y 509.303,Z 778.848,A -85,B 0,C 180,E1 -5495.543,E2 -5495.543} C_VEL
LIN {X 0,Y 509.317,Z 773.837,A -85,B 0,C 180,E1 -5497.133,E2 -5497.133} C_VEL
LIN {X 0,Y 509.483,Z 767.373,A -85,B 0,C 180,E1 -5498.727,E2 -5498.727} C_VEL
LIN {X 0,Y 509.687,Z 759.266,A -85,B 0,C 180,E1 -5500.326,E2 -5500.326} C_VEL
LIN {X 0,Y 509.898,Z 750.521,A -85,B 0,C 180,E1 -5501.748,E2 -5501.748} C_VEL
LIN {X 0,Y 510.311,Z 740.321,A -85,B 0,C 180,E1 -5503.134,E2 -5503.134} C_VEL
LIN {X 0,Y 510.691,Z 729.777,A -85,B 0,C 180,E1 -5504.341,E2 -5504.341} C_VEL
LIN {X 0,Y 511.248,Z 716.867,A -85,B 0,C 180,E1 -5505.582,E2 -5505.582} C_VEL
LIN {X 0,Y 511.775,Z 703.337,A -85,B 0,C 180,E1 -5506.658,E2 -5506.658} C_VEL
LIN {X 0,Y 512.388,Z 689.45,A -85,B 0,C 180,E1 -5507.562,E2 -5507.562} C_VEL
LIN {X 0,Y 512.902,Z 675.1,A -85,B 0,C 180,E1 -5508.318,E2 -5508.318} C_VEL
LIN {X 0,Y 513.407,Z 659.511,A -85,B 0,C 180,E1 -5508.95,E2 -5508.95} C_VEL
LIN {X 0,Y 513.848,Z 644.317,A -85,B 0,C 180,E1 -5509.395,E2 -5509.395} C_VEL
LIN {X 0,Y 514.116,Z 628.274,A -85,B 0,C 180,E1 -5509.697,E2 -5509.697} C_VEL
LIN {X 0,Y 515.193,Z 487.821,A -85,B 0,C 180,E1 -5511.695,E2 -5511.695} C_VEL
LIN {X 0,Y 512.269,Z 467.76,A -85,B 0,C 180,E1 -5512.128,E2 -5512.128} C_VEL
LIN {X 0,Y 513.058,Z 438.478,A -85,B 0,C 180,E1 -5515.127,E2 -5515.127} C_VEL
LIN {X 0,Y 513.783,Z 413.651,A -85,B 0,C 180,E1 -5517.715,E2 -5517.715} C_VEL
LIN {X 0,Y 514.662,Z 386.128,A -85,B 0,C 180,E1 -5520.65,E2 -5520.65} C_VEL
LIN {X 0,Y 510.491,Z 370.102,A -85,B 0,C 180,E1 -5522.674,E2 -5522.674} C_VEL
LIN {X 0,Y 509.834,Z 367.603,A -85,B 0,C 180,E1 -5523.03,E2 -5523.03} C_VEL
LIN {X 0,Y 509.787,Z 367.609,A -85,B 0,C 180,E1 -5525.572,E2 -5525.572} C_VEL
LIN {X 0,Y 509.806,Z 367.609,A -85,B 0,C 180,E1 -5528.34,E2 -5528.34} C_VEL
LIN {X 0,Y 509.82,Z 367.601,A -85,B 0,C 180,E1 -5531.427,E2 -5531.427} C_VEL
LIN {X 0,Y 509.829,Z 367.596,A -85,B 0,C 180,E1 -5534.669,E2 -5534.669} C_VEL
LIN {X 0,Y 509.774,Z 367.606,A -85,B 0,C 180,E1 -5537.504,E2 -5537.504} C_VEL
LIN {X 0,Y 509.819,Z 367.601,A -85,B 0,C 180,E1 -5540.645,E2 -5540.645} C_VEL
LIN {X 0,Y 509.753,Z 367.61,A -85,B 0,C 180,E1 -5543.641,E2 -5543.641} C_VEL
LIN {X 0,Y 509.82,Z 367.606,A -85,B 0,C 180,E1 -5546.536,E2 -5546.536} C_VEL
LIN {X 0,Y 509.814,Z 367.6,A -85,B 0,C 180,E1 -5549.332,E2 -5549.332} C_VEL
LIN {X 0,Y 509.809,Z 367.608,A -85,B 0,C 180,E1 -5552.05,E2 -5552.05} C_VEL
LIN {X 0,Y 509.786,Z 367.608,A -85,B 0,C 180,E1 -5554.699,E2 -5554.699} C_VEL
LIN {X 0,Y 509.809,Z 367.603,A -85,B 0,C 180,E1 -5557.459,E2 -5557.459} C_VEL
LIN {X 0,Y 509.809,Z 367.607,A -85,B 0,C 180,E1 -5560.68,E2 -5560.68} C_VEL
LIN {X 0,Y 509.779,Z 367.606,A -85,B 0,C 180,E1 -5563.171,E2 -5563.171} C_VEL
LIN {X 0,Y 509.824,Z 367.599,A -85,B 0,C 180,E1 -5565.633,E2 -5565.633} C_VEL
LIN {X 0,Y 509.89,Z 367.593,A -85,B 0,C 180,E1 -5568.874,E2 -5568.874} C_VEL
LIN {X 0,Y 509.861,Z 367.598,A -85,B 0,C 180,E1 -5572.077,E2 -5572.077} C_VEL
LIN {X 0,Y 509.916,Z 367.593,A -85,B 0,C 180,E1 -5574.464,E2 -5574.464} C_VEL
LIN {X 0,Y 510.025,Z 367.571,A -85,B 0,C 180,E1 -5577.631,E2 -5577.631} C_VEL
LIN {X 0,Y 510.045,Z 367.575,A -85,B 0,C 180,E1 -5580.79,E2 -5580.79} C_VEL
LIN {X 0,Y 509.895,Z 367.592,A -85,B 0,C 180,E1 -5583.161,E2 -5583.161} C_VEL
LIN {X 0,Y 509.92,Z 367.585,A -85,B 0,C 180,E1 -5586.331,E2 -5586.331} C_VEL
LIN {X 0,Y 509.868,Z 367.595,A -85,B 0,C 180,E1 -5588.721,E2 -5588.721} C_VEL
LIN {X 0,Y 509.89,Z 367.591,A -85,B 0,C 180,E1 -5591.932,E2 -5591.932} C_VEL
LIN {X 0,Y 509.881,Z 367.59,A -85,B 0,C 180,E1 -5595.242,E2 -5595.242} C_VEL
LIN {X 0,Y 509.846,Z 367.602,A -85,B 0,C 180,E1 -5598.485,E2 -5598.485} C_VEL
LIN {X 0,Y 509.836,Z 367.596,A -85,B 0,C 180,E1 -5601.003,E2 -5601.003} C_VEL
LIN {X 0,Y 509.805,Z 367.603,A -85,B 0,C 180,E1 -5603.565,E2 -5603.565} C_VEL
LIN {X 0,Y 509.802,Z 367.602,A -85,B 0,C 180,E1 -5606.357,E2 -5606.357} C_VEL
LIN {X 0,Y 509.836,Z 367.605,A -85,B 0,C 180,E1 -5608.847,E2 -5608.847} C_VEL
LIN {X 0,Y 509.806,Z 367.597,A -85,B 0,C 180,E1 -5611.591,E2 -5611.591} C_VEL
LIN {X 0,Y 509.828,Z 367.603,A -85,B 0,C 180,E1 -5614.416,E2 -5614.416} C_VEL
LIN {X 0,Y 509.806,Z 367.605,A -85,B 0,C 180,E1 -5617.342,E2 -5617.342} C_VEL
LIN {X 0,Y 509.805,Z 367.603,A -85,B 0,C 180,E1 -5620.386,E2 -5620.386} C_VEL
LIN {X 0,Y 509.787,Z 367.608,A -85,B 0,C 180,E1 -5623.06,E2 -5623.06} C_VEL
LIN {X 0,Y 509.815,Z 367.602,A -85,B 0,C 180,E1 -5625.795,E2 -5625.795} C_VEL
LIN {X 0,Y 509.826,Z 367.603,A -85,B 0,C 180,E1 -5628.573,E2 -5628.573} C_VEL
LIN {X 0,Y 509.844,Z 367.596,A -85,B 0,C 180,E1 -5631.788,E2 -5631.788} C_VEL
LIN {X 0,Y 509.8,Z 367.603,A -85,B 0,C 180,E1 -5633.752,E2 -5633.752} C_VEL
LIN {X 0,Y 509.136,Z 367.686,A -85,B 0,C 180,E1 -5634.412,E2 -5634.412} C_VEL
LIN {X 0,Y 506.311,Z 368.043,A -85,B 0,C 180,E1 -5635.483,E2 -5635.483} C_VEL
LIN {X 0,Y 503.915,Z 368.344,A -85,B 0,C 180,E1 -5636.347,E2 -5636.347} C_VEL
LIN {X 0,Y 502.873,Z 368.473,A -85,B 0,C 180,E1 -5637.013,E2 -5637.013} C_VEL
LIN {X 0,Y 502.78,Z 368.481,A -85,B 0,C 180,E1 -5637.239,E2 -5637.239} C_VEL
LIN {X 0,Y 502.824,Z 368.475,A -85,B 0,C 180,E1 -5639.016,E2 -5639.016} C_VEL
LIN {X 0,Y 503.897,Z 371.449,A -85,B 0,C 180,E1 -5639.13,E2 -5639.13} C_VEL
LIN {X 0,Y 508.668,Z 382.314,A -85,B 0,C 180,E1 -5639.526,E2 -5639.526} C_VEL
LIN {X 0,Y 507.813,Z 497.416,A -85,B 0,C 180,E1 -5641.227,E2 -5641.227} C_VEL
LIN {X 0,Y 507.592,Z 512.801,A -85,B 0,C 180,E1 -5641.608,E2 -5641.608} C_VEL
LIN {X 0,Y 507.233,Z 527.719,A -85,B 0,C 180,E1 -5642.148,E2 -5642.148} C_VEL
LIN {X 0,Y 506.765,Z 542.761,A -85,B 0,C 180,E1 -5642.877,E2 -5642.877} C_VEL
LIN {X 0,Y 506.201,Z 556.618,A -85,B 0,C 180,E1 -5643.735,E2 -5643.735} C_VEL
LIN {X 0,Y 505.637,Z 569.942,A -85,B 0,C 180,E1 -5644.759,E2 -5644.759} C_VEL
LIN {X 0,Y 505.033,Z 581.881,A -85,B 0,C 180,E1 -5645.873,E2 -5645.873} C_VEL
LIN {X 0,Y 504.493,Z 592.345,A -85,B 0,C 180,E1 -5647.043,E2 -5647.043} C_VEL
LIN {X 0,Y 503.927,Z 601.931,A -85,B 0,C 180,E1 -5648.311,E2 -5648.311} C_VEL
LIN {X 0,Y 503.536,Z 609.997,A -85,B 0,C 180,E1 -5649.579,E2 -5649.579} C_VEL
LIN {X 0,Y 503.131,Z 617.852,A -85,B 0,C 180,E1 -5651.049,E2 -5651.049} C_VEL
LIN {X 0,Y 502.87,Z 624.288,A -85,B 0,C 180,E1 -5652.514,E2 -5652.514} C_VEL
LIN {X 0,Y 502.648,Z 630.117,A -85,B 0,C 180,E1 -5654.179,E2 -5654.179} C_VEL
LIN {X 0,Y 502.497,Z 633.531,A -85,B 0,C 180,E1 -5655.42,E2 -5655.42} C_VEL
LIN {X 0,Y 502.357,Z 636.944,A -85,B 0,C 180,E1 -5657.066,E2 -5657.066} C_VEL
LIN {X 0,Y 502.357,Z 639.135,A -85,B 0,C 180,E1 -5658.706,E2 -5658.706} C_VEL
LIN {X 0,Y 502.301,Z 640.195,A -85,B 0,C 180,E1 -5660.335,E2 -5660.335} C_VEL
LIN {X 0,Y 502.319,Z 640.137,A -85,B 0,C 180,E1 -5661.958,E2 -5661.958} C_VEL
LIN {X 0,Y 502.403,Z 638.921,A -85,B 0,C 180,E1 -5663.575,E2 -5663.575} C_VEL
LIN {X 0,Y 502.38,Z 636.613,A -85,B 0,C 180,E1 -5665.186,E2 -5665.186} C_VEL
LIN {X 0,Y 502.579,Z 633.128,A -85,B 0,C 180,E1 -5666.794,E2 -5666.794} C_VEL
LIN {X 0,Y 502.623,Z 628.465,A -85,B 0,C 180,E1 -5668.398,E2 -5668.398} C_VEL
LIN {X 0,Y 502.886,Z 622.44,A -85,B 0,C 180,E1 -5670,E2 -5670} C_VEL
LIN {X 0,Y 503.267,Z 614.897,A -85,B 0,C 180,E1 -5671.601,E2 -5671.601} C_VEL
LIN {X 0,Y 503.652,Z 606.893,A -85,B 0,C 180,E1 -5673,E2 -5673} C_VEL
LIN {X 0,Y 504.22,Z 597.257,A -85,B 0,C 180,E1 -5674.397,E2 -5674.397} C_VEL
LIN {X 0,Y 504.721,Z 587.465,A -85,B 0,C 180,E1 -5675.594,E2 -5675.594} C_VEL
LIN {X 0,Y 505.29,Z 575.775,A -85,B 0,C 180,E1 -5676.79,E2 -5676.79} C_VEL
LIN {X 0,Y 505.903,Z 562.805,A -85,B 0,C 180,E1 -5677.885,E2 -5677.885} C_VEL
LIN {X 0,Y 506.493,Z 549.843,A -85,B 0,C 180,E1 -5678.78,E2 -5678.78} C_VEL
LIN {X 0,Y 506.996,Z 535.491,A -85,B 0,C 180,E1 -5679.575,E2 -5679.575} C_VEL
LIN {X 0,Y 507.449,Z 520.416,A -85,B 0,C 180,E1 -5680.215,E2 -5680.215} C_VEL
LIN {X 0,Y 507.673,Z 505.37,A -85,B 0,C 180,E1 -5680.681,E2 -5680.681} C_VEL
LIN {X 0,Y 507.806,Z 490.55,A -85,B 0,C 180,E1 -5680.978,E2 -5680.978} C_VEL
LIN {X 0,Y 508.628,Z 382.193,A -85,B 0,C 180,E1 -5682.557,E2 -5682.557} C_VEL
LIN {X 0,Y 502.875,Z 369.026,A -85,B 0,C 180,E1 -5683.023,E2 -5683.023} C_VEL
LIN {X 0,Y 502.787,Z 368.484,A -85,B 0,C 180,E1 -5683.062,E2 -5683.062} C_VEL
LIN {X 0,Y 502.793,Z 368.48,A -85,B 0,C 180,E1 -5685.401,E2 -5685.401} C_VEL
LIN {X 0,Y 502.799,Z 368.481,A -85,B 0,C 180,E1 -5688.753,E2 -5688.753} C_VEL
LIN {X 0,Y 502.764,Z 368.484,A -85,B 0,C 180,E1 -5691.312,E2 -5691.312} C_VEL
LIN {X 0,Y 502.739,Z 368.483,A -85,B 0,C 180,E1 -5693.916,E2 -5693.916} C_VEL
LIN {X 0,Y 502.757,Z 368.484,A -85,B 0,C 180,E1 -5696.572,E2 -5696.572} C_VEL
LIN {X 0,Y 502.751,Z 368.48,A -85,B 0,C 180,E1 -5699.292,E2 -5699.292} C_VEL
LIN {X 0,Y 502.754,Z 368.481,A -85,B 0,C 180,E1 -5702.086,E2 -5702.086} C_VEL
LIN {X 0,Y 502.778,Z 368.483,A -85,B 0,C 180,E1 -5704.967,E2 -5704.967} C_VEL
LIN {X 0,Y 502.753,Z 368.482,A -85,B 0,C 180,E1 -5708.479,E2 -5708.479} C_VEL
LIN {X 0,Y 502.754,Z 368.485,A -85,B 0,C 180,E1 -5711.072,E2 -5711.072} C_VEL
LIN {X 0,Y 502.774,Z 368.477,A -85,B 0,C 180,E1 -5714.528,E2 -5714.528} C_VEL
LIN {X 0,Y 502.761,Z 368.479,A -85,B 0,C 180,E1 -5717.857,E2 -5717.857} C_VEL
LIN {X 0,Y 502.771,Z 368.484,A -85,B 0,C 180,E1 -5721.021,E2 -5721.021} C_VEL
LIN {X 0,Y 502.758,Z 368.48,A -85,B 0,C 180,E1 -5724.17,E2 -5724.17} C_VEL
LIN {X 0,Y 502.762,Z 368.481,A -85,B 0,C 180,E1 -5727.004,E2 -5727.004} C_VEL
LIN {X 0,Y 502.739,Z 368.481,A -85,B 0,C 180,E1 -5730.078,E2 -5730.078} C_VEL
LIN {X 0,Y 502.76,Z 368.479,A -85,B 0,C 180,E1 -5732.529,E2 -5732.529} C_VEL
LIN {X 0,Y 502.754,Z 368.486,A -85,B 0,C 180,E1 -5735.315,E2 -5735.315} C_VEL
LIN {X 0,Y 502.77,Z 368.481,A -85,B 0,C 180,E1 -5737.826,E2 -5737.826} C_VEL
LIN {X 0,Y 502.801,Z 368.472,A -85,B 0,C 180,E1 -5740.399,E2 -5740.399} C_VEL
LIN {X 0,Y 502.788,Z 368.477,A -85,B 0,C 180,E1 -5742.93,E2 -5742.93} C_VEL
LIN {X 0,Y 502.817,Z 368.477,A -85,B 0,C 180,E1 -5745.428,E2 -5745.428} C_VEL
LIN {X 0,Y 502.861,Z 368.453,A -85,B 0,C 180,E1 -5748.716,E2 -5748.716} C_VEL
LIN {X 0,Y 502.835,Z 368.469,A -85,B 0,C 180,E1 -5751.965,E2 -5751.965} C_VEL
LIN {X 0,Y 502.884,Z 368.464,A -85,B 0,C 180,E1 -5754.386,E2 -5754.386} C_VEL
LIN {X 0,Y 502.993,Z 368.452,A -85,B 0,C 180,E1 -5757.597,E2 -5757.597} C_VEL
LIN {X 0,Y 502.985,Z 368.453,A -85,B 0,C 180,E1 -5760,E2 -5760} C_VEL
LIN {X 0,Y 502.998,Z 368.448,A -85,B 0,C 180,E1 -5762.402,E2 -5762.402} C_VEL
LIN {X 0,Y 502.874,Z 368.472,A -85,B 0,C 180,E1 -5765.614,E2 -5765.614} C_VEL
LIN {X 0,Y 502.837,Z 368.47,A -85,B 0,C 180,E1 -5768.034,E2 -5768.034} C_VEL
LIN {X 0,Y 502.862,Z 368.47,A -85,B 0,C 180,E1 -5771.283,E2 -5771.283} C_VEL
LIN {X 0,Y 502.812,Z 368.47,A -85,B 0,C 180,E1 -5774.572,E2 -5774.572} C_VEL
LIN {X 0,Y 502.772,Z 368.481,A -85,B 0,C 180,E1 -5777.91,E2 -5777.91} C_VEL
LIN {X 0,Y 502.792,Z 368.476,A -85,B 0,C 180,E1 -5780.528,E2 -5780.528} C_VEL
LIN {X 0,Y 502.771,Z 368.477,A -85,B 0,C 180,E1 -5783.041,E2 -5783.041} C_VEL
LIN {X 0,Y 502.766,Z 368.486,A -85,B 0,C 180,E1 -5785.679,E2 -5785.679} C_VEL
LIN {X 0,Y 502.76,Z 368.48,A -85,B 0,C 180,E1 -5788.377,E2 -5788.377} C_VEL
LIN {X 0,Y 502.776,Z 368.48,A -85,B 0,C 180,E1 -5791.144,E2 -5791.144} C_VEL
LIN {X 0,Y 502.775,Z 368.48,A -85,B 0,C 180,E1 -5793.996,E2 -5793.996} C_VEL
LIN {X 0,Y 502.722,Z 368.487,A -85,B 0,C 180,E1 -5797.171,E2 -5797.171} C_VEL
LIN {X 0,Y 502.761,Z 368.486,A -85,B 0,C 180,E1 -5800.018,E2 -5800.018} C_VEL
LIN {X 0,Y 502.73,Z 368.483,A -85,B 0,C 180,E1 -5803.236,E2 -5803.236} C_VEL
LIN {X 0,Y 502.772,Z 368.482,A -85,B 0,C 180,E1 -5805.66,E2 -5805.66} C_VEL
LIN {X 0,Y 502.745,Z 368.476,A -85,B 0,C 180,E1 -5809.015,E2 -5809.015} C_VEL
LIN {X 0,Y 502.753,Z 368.488,A -85,B 0,C 180,E1 -5812.043,E2 -5812.043} C_VEL
LIN {X 0,Y 502.778,Z 368.481,A -85,B 0,C 180,E1 -5815.033,E2 -5815.033} C_VEL
LIN {X 0,Y 502.818,Z 368.622,A -85,B 0,C 180,E1 -5816.795,E2 -5816.795} C_VEL
LIN {X 0,Y 507.876,Z 387.905,A -85,B 0,C 180,E1 -5819.203,E2 -5819.203} C_VEL
LIN {X 0,Y 507.083,Z 411.903,A -85,B 0,C 180,E1 -5821.774,E2 -5821.774} C_VEL
LIN {X 0,Y 506.28,Z 438.431,A -85,B 0,C 180,E1 -5824.578,E2 -5824.578} C_VEL
LIN {X 0,Y 505.44,Z 467.034,A -85,B 0,C 180,E1 -5827.562,E2 -5827.562} C_VEL
LIN {X 0,Y 508.524,Z 487.827,A -85,B 0,C 180,E1 -5828.018,E2 -5828.018} C_VEL
LIN {X 0,Y 507.342,Z 635.175,A -85,B 0,C 180,E1 -5830.161,E2 -5830.161} C_VEL
LIN {X 0,Y 506.87,Z 651.152,A -85,B 0,C 180,E1 -5830.543,E2 -5830.543} C_VEL
LIN {X 0,Y 506.377,Z 666.998,A -85,B 0,C 180,E1 -5831.106,E2 -5831.106} C_VEL
LIN {X 0,Y 505.798,Z 681.322,A -85,B 0,C 180,E1 -5831.782,E2 -5831.782} C_VEL
LIN {X 0,Y 505.215,Z 695.055,A -85,B 0,C 180,E1 -5832.598,E2 -5832.598} C_VEL
LIN {X 0,Y 504.609,Z 709.073,A -85,B 0,C 180,E1 -5833.618,E2 -5833.618} C_VEL
LIN {X 0,Y 503.973,Z 721.788,A -85,B 0,C 180,E1 -5834.739,E2 -5834.739} C_VEL
LIN {X 0,Y 503.471,Z 734.314,A -85,B 0,C 180,E1 -5836.067,E2 -5836.067} C_VEL
LIN {X 0,Y 503.031,Z 745.477,A -85,B 0,C 180,E1 -5837.493,E2 -5837.493} C_VEL
LIN {X 0,Y 502.762,Z 754.803,A -85,B 0,C 180,E1 -5838.918,E2 -5838.918} C_VEL
LIN {X 0,Y 502.454,Z 762.537,A -85,B 0,C 180,E1 -5840.337,E2 -5840.337} C_VEL
LIN {X 0,Y 502.34,Z 769.792,A -85,B 0,C 180,E1 -5841.958,E2 -5841.958} C_VEL
LIN {X 0,Y 502.233,Z 775.501,A -85,B 0,C 180,E1 -5843.572,E2 -5843.572} C_VEL
LIN {X 0,Y 502.137,Z 779.818,A -85,B 0,C 180,E1 -5845.183,E2 -5845.183} C_VEL
LIN {X 0,Y 502.148,Z 782.856,A -85,B 0,C 180,E1 -5846.79,E2 -5846.79} C_VEL
LIN {X 0,Y 502.08,Z 784.657,A -85,B 0,C 180,E1 -5848.395,E2 -5848.395} C_VEL
LIN {X 0,Y 502.057,Z 785.272,A -85,B 0,C 180,E1 -5850,E2 -5850} C_VEL
LIN {X 0,Y 502.081,Z 784.651,A -85,B 0,C 180,E1 -5851.604,E2 -5851.604} C_VEL
LIN {X 0,Y 502.149,Z 782.842,A -85,B 0,C 180,E1 -5853.209,E2 -5853.209} C_VEL
LIN {X 0,Y 502.136,Z 779.799,A -85,B 0,C 180,E1 -5854.817,E2 -5854.817} C_VEL
LIN {X 0,Y 502.232,Z 775.479,A -85,B 0,C 180,E1 -5856.427,E2 -5856.427} C_VEL
LIN {X 0,Y 502.34,Z 769.756,A -85,B 0,C 180,E1 -5858.042,E2 -5858.042} C_VEL
LIN {X 0,Y 502.455,Z 762.479,A -85,B 0,C 180,E1 -5859.662,E2 -5859.662} C_VEL
LIN {X 0,Y 502.752,Z 754.729,A -85,B 0,C 180,E1 -5861.081,E2 -5861.081} C_VEL
LIN {X 0,Y 503.039,Z 745.392,A -85,B 0,C 180,E1 -5862.506,E2 -5862.506} C_VEL
LIN {X 0,Y 503.471,Z 734.204,A -85,B 0,C 180,E1 -5863.933,E2 -5863.933} C_VEL
LIN {X 0,Y 503.96,Z 721.659,A -85,B 0,C 180,E1 -5865.261,E2 -5865.261} C_VEL
LIN {X 0,Y 504.607,Z 708.929,A -85,B 0,C 180,E1 -5866.381,E2 -5866.381} C_VEL
LIN {X 0,Y 505.189,Z 694.871,A -85,B 0,C 180,E1 -5867.403,E2 -5867.403} C_VEL
LIN {X 0,Y 505.763,Z 681.113,A -85,B 0,C 180,E1 -5868.219,E2 -5868.219} C_VEL
LIN {X 0,Y 506.336,Z 666.688,A -85,B 0,C 180,E1 -5868.899,E2 -5868.899} C_VEL
LIN {X 0,Y 506.881,Z 651.117,A -85,B 0,C 180,E1 -5869.451,E2 -5869.451} C_VEL
LIN {X 0,Y 507.338,Z 634.955,A -85,B 0,C 180,E1 -5869.838,E2 -5869.838} C_VEL
LIN {X 0,Y 508.511,Z 487.805,A -85,B 0,C 180,E1 -5871.979,E2 -5871.979} C_VEL
LIN {X 0,Y 505.397,Z 466.788,A -85,B 0,C 180,E1 -5872.432,E2 -5872.432} C_VEL
LIN {X 0,Y 506.325,Z 435.598,A -85,B 0,C 180,E1 -5875.683,E2 -5875.683} C_VEL
LIN {X 0,Y 506.995,Z 412.711,A -85,B 0,C 180,E1 -5878.118,E2 -5878.118} C_VEL
LIN {X 0,Y 507.926,Z 389.006,A -85,B 0,C 180,E1 -5880.685,E2 -5880.685} C_VEL
LIN {X 0,Y 506.649,Z 382.739,A -85,B 0,C 180,E1 -5881.459,E2 -5881.459} C_VEL
LIN {X 0,Y 502.807,Z 368.48,A -85,B 0,C 180,E1 -5883.33,E2 -5883.33} C_VEL
LIN {X 0,Y 502.737,Z 368.484,A -85,B 0,C 180,E1 -5885.953,E2 -5885.953} C_VEL
LIN {X 0,Y 502.774,Z 368.48,A -85,B 0,C 180,E1 -5888.977,E2 -5888.977} C_VEL
LIN {X 0,Y 502.762,Z 368.485,A -85,B 0,C 180,E1 -5892.194,E2 -5892.194} C_VEL
LIN {X 0,Y 502.767,Z 368.474,A -85,B 0,C 180,E1 -5895.47,E2 -5895.47} C_VEL
LIN {X 0,Y 502.751,Z 368.481,A -85,B 0,C 180,E1 -5898.927,E2 -5898.927} C_VEL
LIN {X 0,Y 502.747,Z 368.485,A -85,B 0,C 180,E1 -5902.042,E2 -5902.042} C_VEL
LIN {X 0,Y 502.769,Z 368.48,A -85,B 0,C 180,E1 -5905.032,E2 -5905.032} C_VEL
LIN {X 0,Y 502.75,Z 368.485,A -85,B 0,C 180,E1 -5907.913,E2 -5907.913} C_VEL
LIN {X 0,Y 502.788,Z 368.481,A -85,B 0,C 180,E1 -5910.71,E2 -5910.71} C_VEL
LIN {X 0,Y 502.759,Z 368.48,A -85,B 0,C 180,E1 -5913.459,E2 -5913.459} C_VEL
LIN {X 0,Y 502.745,Z 368.486,A -85,B 0,C 180,E1 -5916.084,E2 -5916.084} C_VEL
LIN {X 0,Y 502.743,Z 368.485,A -85,B 0,C 180,E1 -5918.687,E2 -5918.687} C_VEL
LIN {X 0,Y 502.777,Z 368.481,A -85,B 0,C 180,E1 -5921.897,E2 -5921.897} C_VEL
LIN {X 0,Y 502.82,Z 368.477,A -85,B 0,C 180,E1 -5924.665,E2 -5924.665} C_VEL
LIN {X 0,Y 502.861,Z 368.47,A -85,B 0,C 180,E1 -5928.039,E2 -5928.039} C_VEL
LIN {X 0,Y 502.824,Z 368.473,A -85,B 0,C 180,E1 -5931.156,E2 -5931.156} C_VEL
LIN {X 0,Y 502.832,Z 368.467,A -85,B 0,C 180,E1 -5933.58,E2 -5933.58} C_VEL
LIN {X 0,Y 502.848,Z 368.47,A -85,B 0,C 180,E1 -5936.795,E2 -5936.795} C_VEL
LIN {X 0,Y 502.885,Z 368.467,A -85,B 0,C 180,E1 -5938.399,E2 -5938.399} C_VEL
LIN {X 0,Y 502.994,Z 368.453,A -85,B 0,C 180,E1 -5940.801,E2 -5940.801} C_VEL
LIN {X 0,Y 502.995,Z 368.454,A -85,B 0,C 180,E1 -5942.403,E2 -5942.403} C_VEL
LIN {X 0,Y 502.903,Z 368.456,A -85,B 0,C 180,E1 -5945.614,E2 -5945.614} C_VEL
LIN {X 0,Y 502.857,Z 368.458,A -85,B 0,C 180,E1 -5948.034,E2 -5948.034} C_VEL
LIN {X 0,Y 502.858,Z 368.468,A -85,B 0,C 180,E1 -5951.284,E2 -5951.284} C_VEL
LIN {X 0,Y 502.817,Z 368.468,A -85,B 0,C 180,E1 -5954.572,E2 -5954.572} C_VEL
LIN {X 0,Y 502.802,Z 368.478,A -85,B 0,C 180,E1 -5957.07,E2 -5957.07} C_VEL
LIN {X 0,Y 502.808,Z 368.469,A -85,B 0,C 180,E1 -5959.601,E2 -5959.601} C_VEL
LIN {X 0,Y 502.789,Z 368.479,A -85,B 0,C 180,E1 -5962.703,E2 -5962.703} C_VEL
LIN {X 0,Y 502.763,Z 368.476,A -85,B 0,C 180,E1 -5965.68,E2 -5965.68} C_VEL
LIN {X 0,Y 502.765,Z 368.479,A -85,B 0,C 180,E1 -5968.378,E2 -5968.378} C_VEL
LIN {X 0,Y 502.782,Z 368.476,A -85,B 0,C 180,E1 -5971.145,E2 -5971.145} C_VEL
LIN {X 0,Y 502.779,Z 368.479,A -85,B 0,C 180,E1 -5973.996,E2 -5973.996} C_VEL
LIN {X 0,Y 502.767,Z 368.483,A -85,B 0,C 180,E1 -5977.179,E2 -5977.179} C_VEL
LIN {X 0,Y 502.762,Z 368.478,A -85,B 0,C 180,E1 -5980.018,E2 -5980.018} C_VEL
LIN {X 0,Y 502.742,Z 368.483,A -85,B 0,C 180,E1 -5983.235,E2 -5983.235} C_VEL
LIN {X 0,Y 502.772,Z 368.48,A -85,B 0,C 180,E1 -5985.661,E2 -5985.661} C_VEL
LIN {X 0,Y 502.789,Z 368.477,A -85,B 0,C 180,E1 -5987.862,E2 -5987.862} C_VEL
LIN {X 0,Y 502.787,Z 368.485,A -85,B 0,C 180,E1 -5991.024,E2 -5991.024} C_VEL
LIN {X 0,Y 502.765,Z 368.478,A -85,B 0,C 180,E1 -5994.171,E2 -5994.171} C_VEL
LIN {X 0,Y 502.78,Z 368.481,A -85,B 0,C 180,E1 -5997.239,E2 -5997.239} C_VEL
LIN {X 0,Y 502.735,Z 369.186,A -85,B 0,C 180,E1 -5997.66,E2 -5997.66} C_VEL
LIN {X 0,Y 502.664,Z 370.953,A -85,B 0,C 180,E1 -5998.043,E2 -5998.043} C_VEL
LIN {X 0,Y 502.534,Z 374.914,A -85,B 0,C 180,E1 -5998.532,E2 -5998.532} C_VEL
LIN {X 0,Y 502.387,Z 380.016,A -85,B 0,C 180,E1 -5998.917,E2 -5998.917} C_VEL
LIN {X 0,Y 502.243,Z 385.762,A -85,B 0,C 180,E1 -5999.197,E2 -5999.197} C_VEL
LIN {X 0,Y 502.126,Z 391.852,A -85,B 0,C 180,E1 -5999.354,E2 -5999.354} C_VEL
LIN {X 0,Y 501.189,Z 498.684,A -85,B 0,C 180,E1 -6000.954,E2 -6000.954} C_VEL
LIN {X 0,Y 500.982,Z 513.983,A -85,B 0,C 180,E1 -6001.342,E2 -6001.342} C_VEL
LIN {X 0,Y 500.599,Z 528.883,A -85,B 0,C 180,E1 -6001.89,E2 -6001.89} C_VEL
LIN {X 0,Y 500.119,Z 543.327,A -85,B 0,C 180,E1 -6002.6,E2 -6002.6} C_VEL
LIN {X 0,Y 499.52,Z 557.269,A -85,B 0,C 180,E1 -6003.469,E2 -6003.469} C_VEL
LIN {X 0,Y 498.918,Z 570.641,A -85,B 0,C 180,E1 -6004.504,E2 -6004.504} C_VEL
LIN {X 0,Y 498.274,Z 582.65,A -85,B 0,C 180,E1 -6005.635,E2 -6005.635} C_VEL
LIN {X 0,Y 497.663,Z 594.05,A -85,B 0,C 180,E1 -6006.929,E2 -6006.929} C_VEL
LIN {X 0,Y 497.044,Z 603.524,A -85,B 0,C 180,E1 -6008.213,E2 -6008.213} C_VEL
LIN {X 0,Y 496.562,Z 612.723,A -85,B 0,C 180,E1 -6009.712,E2 -6009.712} C_VEL
LIN {X 0,Y 496.191,Z 619.257,A -85,B 0,C 180,E1 -6010.989,E2 -6010.989} C_VEL
LIN {X 0,Y 495.856,Z 626.413,A -85,B 0,C 180,E1 -6012.685,E2 -6012.685} C_VEL
LIN {X 0,Y 495.639,Z 631.979,A -85,B 0,C 180,E1 -6014.371,E2 -6014.371} C_VEL
LIN {X 0,Y 495.433,Z 636.145,A -85,B 0,C 180,E1 -6016.046,E2 -6016.046} C_VEL
LIN {X 0,Y 495.306,Z 639.042,A -85,B 0,C 180,E1 -6017.712,E2 -6017.712} C_VEL
LIN {X 0,Y 495.265,Z 640.757,A -85,B 0,C 180,E1 -6019.37,E2 -6019.37} C_VEL
LIN {X 0,Y 495.302,Z 641.33,A -85,B 0,C 180,E1 -6021.021,E2 -6021.021} C_VEL
LIN {X 0,Y 495.34,Z 640.751,A -85,B 0,C 180,E1 -6022.664,E2 -6022.664} C_VEL
LIN {X 0,Y 495.378,Z 639.081,A -85,B 0,C 180,E1 -6024.301,E2 -6024.301} C_VEL
LIN {X 0,Y 495.4,Z 636.304,A -85,B 0,C 180,E1 -6025.933,E2 -6025.933} C_VEL
LIN {X 0,Y 495.589,Z 632.33,A -85,B 0,C 180,E1 -6027.562,E2 -6027.562} C_VEL
LIN {X 0,Y 495.772,Z 627.108,A -85,B 0,C 180,E1 -6029.188,E2 -6029.188} C_VEL
LIN {X 0,Y 496.128,Z 620.465,A -85,B 0,C 180,E1 -6030.812,E2 -6030.812} C_VEL
LIN {X 0,Y 496.558,Z 612.213,A -85,B 0,C 180,E1 -6032.434,E2 -6032.434} C_VEL
LIN {X 0,Y 497.041,Z 603.469,A -85,B 0,C 180,E1 -6033.851,E2 -6033.851} C_VEL
LIN {X 0,Y 497.687,Z 592.917,A -85,B 0,C 180,E1 -6035.267,E2 -6035.267} C_VEL
LIN {X 0,Y 498.22,Z 582.135,A -85,B 0,C 180,E1 -6036.48,E2 -6036.48} C_VEL
LIN {X 0,Y 498.846,Z 570.298,A -85,B 0,C 180,E1 -6037.59,E2 -6037.59} C_VEL
LIN {X 0,Y 499.508,Z 557.254,A -85,B 0,C 180,E1 -6038.598,E2 -6038.598} C_VEL
LIN {X 0,Y 500.03,Z 544.48,A -85,B 0,C 180,E1 -6039.404,E2 -6039.404} C_VEL
LIN {X 0,Y 500.543,Z 529.903,A -85,B 0,C 180,E1 -6040.135,E2 -6040.135} C_VEL
LIN {X 0,Y 500.891,Z 514.59,A -85,B 0,C 180,E1 -6040.714,E2 -6040.714} C_VEL
LIN {X 0,Y 501.108,Z 499.012,A -85,B 0,C 180,E1 -6041.119,E2 -6041.119} C_VEL
LIN {X 0,Y 502.037,Z 384.054,A -85,B 0,C 180,E1 -6042.835,E2 -6042.835} C_VEL
LIN {X 0,Y 495.849,Z 369.928,A -85,B 0,C 180,E1 -6043.342,E2 -6043.342} C_VEL
LIN {X 0,Y 495.74,Z 369.361,A -85,B 0,C 180,E1 -6043.365,E2 -6043.365} C_VEL
LIN {X 0,Y 495.731,Z 369.359,A -85,B 0,C 180,E1 -6046.472,E2 -6046.472} C_VEL
LIN {X 0,Y 495.752,Z 369.359,A -85,B 0,C 180,E1 -6049.03,E2 -6049.03} C_VEL
LIN {X 0,Y 495.729,Z 369.358,A -85,B 0,C 180,E1 -6051.629,E2 -6051.629} C_VEL
LIN {X 0,Y 495.692,Z 369.362,A -85,B 0,C 180,E1 -6054.278,E2 -6054.278} C_VEL
LIN {X 0,Y 495.717,Z 369.364,A -85,B 0,C 180,E1 -6056.979,E2 -6056.979} C_VEL
LIN {X 0,Y 495.694,Z 369.353,A -85,B 0,C 180,E1 -6059.751,E2 -6059.751} C_VEL
LIN {X 0,Y 495.723,Z 369.359,A -85,B 0,C 180,E1 -6062.597,E2 -6062.597} C_VEL
LIN {X 0,Y 495.725,Z 369.359,A -85,B 0,C 180,E1 -6065.539,E2 -6065.539} C_VEL
LIN {X 0,Y 495.729,Z 369.359,A -85,B 0,C 180,E1 -6068.763,E2 -6068.763} C_VEL
LIN {X 0,Y 495.719,Z 369.358,A -85,B 0,C 180,E1 -6071.784,E2 -6071.784} C_VEL
LIN {X 0,Y 495.727,Z 369.362,A -85,B 0,C 180,E1 -6075.141,E2 -6075.141} C_VEL
LIN {X 0,Y 495.718,Z 369.355,A -85,B 0,C 180,E1 -6078.215,E2 -6078.215} C_VEL
LIN {X 0,Y 495.728,Z 369.361,A -85,B 0,C 180,E1 -6081.236,E2 -6081.236} C_VEL
LIN {X 0,Y 495.731,Z 369.356,A -85,B 0,C 180,E1 -6084.461,E2 -6084.461} C_VEL
LIN {X 0,Y 495.717,Z 369.365,A -85,B 0,C 180,E1 -6087.402,E2 -6087.402} C_VEL
LIN {X 0,Y 495.691,Z 369.358,A -85,B 0,C 180,E1 -6090.248,E2 -6090.248} C_VEL
LIN {X 0,Y 495.712,Z 369.365,A -85,B 0,C 180,E1 -6093.274,E2 -6093.274} C_VEL
LIN {X 0,Y 495.694,Z 369.36,A -85,B 0,C 180,E1 -6095.722,E2 -6095.722} C_VEL
LIN {X 0,Y 495.731,Z 369.355,A -85,B 0,C 180,E1 -6098.37,E2 -6098.37} C_VEL
LIN {X 0,Y 495.758,Z 369.353,A -85,B 0,C 180,E1 -6100.97,E2 -6100.97} C_VEL
LIN {X 0,Y 495.814,Z 369.344,A -85,B 0,C 180,E1 -6104.549,E2 -6104.549} C_VEL
LIN {X 0,Y 495.819,Z 369.331,A -85,B 0,C 180,E1 -6107.965,E2 -6107.965} C_VEL
LIN {X 0,Y 495.767,Z 369.341,A -85,B 0,C 180,E1 -6111.029,E2 -6111.029} C_VEL
LIN {X 0,Y 495.808,Z 369.351,A -85,B 0,C 180,E1 -6113.489,E2 -6113.489} C_VEL
LIN {X 0,Y 495.681,Z 369.362,A -85,B 0,C 180,E1 -6115.935,E2 -6115.935} C_VEL
LIN {X 0,Y 495.96,Z 369.328,A -85,B 0,C 180,E1 -6117.563,E2 -6117.563} C_VEL
LIN {X 0,Y 495.955,Z 369.329,A -85,B 0,C 180,E1 -6120,E2 -6120} C_VEL
LIN {X 0,Y 495.967,Z 369.323,A -85,B 0,C 180,E1 -6122.436,E2 -6122.436} C_VEL
LIN {X 0,Y 495.831,Z 369.349,A -85,B 0,C 180,E1 -6125.694,E2 -6125.694} C_VEL
LIN {X 0,Y 495.8,Z 369.345,A -85,B 0,C 180,E1 -6128.149,E2 -6128.149} C_VEL
LIN {X 0,Y 495.838,Z 369.347,A -85,B 0,C 180,E1 -6131.445,E2 -6131.445} C_VEL
LIN {X 0,Y 495.763,Z 369.348,A -85,B 0,C 180,E1 -6134.783,E2 -6134.783} C_VEL
LIN {X 0,Y 495.737,Z 369.353,A -85,B 0,C 180,E1 -6138.226,E2 -6138.226} C_VEL
LIN {X 0,Y 495.736,Z 369.355,A -85,B 0,C 180,E1 -6140.758,E2 -6140.758} C_VEL
LIN {X 0,Y 495.724,Z 369.358,A -85,B 0,C 180,E1 -6143.388,E2 -6143.388} C_VEL
LIN {X 0,Y 495.707,Z 369.361,A -85,B 0,C 180,E1 -6146.072,E2 -6146.072} C_VEL
LIN {X 0,Y 495.715,Z 369.357,A -85,B 0,C 180,E1 -6148.818,E2 -6148.818} C_VEL
LIN {X 0,Y 495.733,Z 369.363,A -85,B 0,C 180,E1 -6151.723,E2 -6151.723} C_VEL
LIN {X 0,Y 495.746,Z 369.352,A -85,B 0,C 180,E1 -6154.692,E2 -6154.692} C_VEL
LIN {X 0,Y 495.689,Z 369.367,A -85,B 0,C 180,E1 -6157.565,E2 -6157.565} C_VEL
LIN {X 0,Y 495.733,Z 369.361,A -85,B 0,C 180,E1 -6160.045,E2 -6160.045} C_VEL
LIN {X 0,Y 495.682,Z 369.36,A -85,B 0,C 180,E1 -6162.888,E2 -6162.888} C_VEL
LIN {X 0,Y 495.716,Z 369.363,A -85,B 0,C 180,E1 -6165.998,E2 -6165.998} C_VEL
LIN {X 0,Y 495.704,Z 369.353,A -85,B 0,C 180,E1 -6169.295,E2 -6169.295} C_VEL
LIN {X 0,Y 495.714,Z 369.361,A -85,B 0,C 180,E1 -6171.406,E2 -6171.406} C_VEL
LIN {X 0,Y 495.723,Z 369.361,A -85,B 0,C 180,E1 -6174.461,E2 -6174.461} C_VEL
LIN {X 0,Y 495.793,Z 369.536,A -85,B 0,C 180,E1 -6176.513,E2 -6176.513} C_VEL
LIN {X 0,Y 500.724,Z 388.262,A -85,B 0,C 180,E1 -6178.89,E2 -6178.89} C_VEL
LIN {X 0,Y 501.109,Z 390.013,A -85,B 0,C 180,E1 -6179.103,E2 -6179.103} C_VEL
LIN {X 0,Y 500.151,Z 416.425,A -85,B 0,C 180,E1 -6181.964,E2 -6181.964} C_VEL
LIN {X 0,Y 499.326,Z 441.204,A -85,B 0,C 180,E1 -6184.612,E2 -6184.612} C_VEL
LIN {X 0,Y 498.57,Z 466.103,A -85,B 0,C 180,E1 -6187.246,E2 -6187.246} C_VEL
LIN {X 0,Y 501.919,Z 489.604,A -85,B 0,C 180,E1 -6187.755,E2 -6187.755} C_VEL
LIN {X 0,Y 500.612,Z 635.513,A -85,B 0,C 180,E1 -6189.909,E2 -6189.909} C_VEL
LIN {X 0,Y 500.085,Z 651.524,A -85,B 0,C 180,E1 -6190.314,E2 -6190.314} C_VEL
LIN {X 0,Y 499.535,Z 666.518,A -85,B 0,C 180,E1 -6190.862,E2 -6190.862} C_VEL
LIN {X 0,Y 499.013,Z 680.298,A -85,B 0,C 180,E1 -6191.525,E2 -6191.525} C_VEL
LIN {X 0,Y 498.355,Z 694.027,A -85,B 0,C 180,E1 -6192.35,E2 -6192.35} C_VEL
LIN {X 0,Y 497.655,Z 708.039,A -85,B 0,C 180,E1 -6193.383,E2 -6193.383} C_VEL
LIN {X 0,Y 497.016,Z 720.76,A -85,B 0,C 180,E1 -6194.52,E2 -6194.52} C_VEL
LIN {X 0,Y 496.453,Z 733.284,A -85,B 0,C 180,E1 -6195.866,E2 -6195.866} C_VEL
LIN {X 0,Y 495.997,Z 744.45,A -85,B 0,C 180,E1 -6197.313,E2 -6197.313} C_VEL
LIN {X 0,Y 495.709,Z 753.778,A -85,B 0,C 180,E1 -6198.759,E2 -6198.759} C_VEL
LIN {X 0,Y 495.394,Z 761.514,A -85,B 0,C 180,E1 -6200.198,E2 -6200.198} C_VEL
LIN {X 0,Y 495.287,Z 768.774,A -85,B 0,C 180,E1 -6201.842,E2 -6201.842} C_VEL
LIN {X 0,Y 495.201,Z 774.488,A -85,B 0,C 180,E1 -6203.481,E2 -6203.481} C_VEL
LIN {X 0,Y 495.113,Z 778.808,A -85,B 0,C 180,E1 -6205.114,E2 -6205.114} C_VEL
LIN {X 0,Y 495.107,Z 781.844,A -85,B 0,C 180,E1 -6206.745,E2 -6206.745} C_VEL
LIN {X 0,Y 495.051,Z 783.645,A -85,B 0,C 180,E1 -6208.373,E2 -6208.373} C_VEL
LIN {X 0,Y 495.051,Z 784.261,A -85,B 0,C 180,E1 -6210,E2 -6210} C_VEL
LIN {X 0,Y 495.052,Z 783.633,A -85,B 0,C 180,E1 -6211.627,E2 -6211.627} C_VEL
LIN {X 0,Y 495.11,Z 781.82,A -85,B 0,C 180,E1 -6213.255,E2 -6213.255} C_VEL
LIN {X 0,Y 495.112,Z 778.774,A -85,B 0,C 180,E1 -6214.885,E2 -6214.885} C_VEL
LIN {X 0,Y 495.201,Z 774.316,A -85,B 0,C 180,E1 -6216.56,E2 -6216.56} C_VEL
LIN {X 0,Y 495.287,Z 768.714,A -85,B 0,C 180,E1 -6218.157,E2 -6218.157} C_VEL
LIN {X 0,Y 495.395,Z 761.428,A -85,B 0,C 180,E1 -6219.801,E2 -6219.801} C_VEL
LIN {X 0,Y 495.697,Z 753.672,A -85,B 0,C 180,E1 -6221.241,E2 -6221.241} C_VEL
LIN {X 0,Y 495.998,Z 744.328,A -85,B 0,C 180,E1 -6222.686,E2 -6222.686} C_VEL
LIN {X 0,Y 496.455,Z 733.134,A -85,B 0,C 180,E1 -6224.134,E2 -6224.134} C_VEL
LIN {X 0,Y 497.005,Z 720.588,A -85,B 0,C 180,E1 -6225.479,E2 -6225.479} C_VEL
LIN {X 0,Y 497.642,Z 707.847,A -85,B 0,C 180,E1 -6226.617,E2 -6226.617} C_VEL
LIN {X 0,Y 498.328,Z 693.795,A -85,B 0,C 180,E1 -6227.65,E2 -6227.65} C_VEL
LIN {X 0,Y 498.945,Z 680.033,A -85,B 0,C 180,E1 -6228.476,E2 -6228.476} C_VEL
LIN {X 0,Y 499.59,Z 665.105,A -85,B 0,C 180,E1 -6229.185,E2 -6229.185} C_VEL
LIN {X 0,Y 500.169,Z 649.633,A -85,B 0,C 180,E1 -6229.734,E2 -6229.734} C_VEL
LIN {X 0,Y 500.616,Z 633.824,A -85,B 0,C 180,E1 -6230.117,E2 -6230.117} C_VEL
LIN {X 0,Y 501.929,Z 489.416,A -85,B 0,C 180,E1 -6232.242,E2 -6232.242} C_VEL
LIN {X 0,Y 498.48,Z 465.529,A -85,B 0,C 180,E1 -6232.78,E2 -6232.78} C_VEL
LIN {X 0,Y 499.494,Z 435.444,A -85,B 0,C 180,E1 -6235.971,E2 -6235.971} C_VEL
LIN {X 0,Y 500.396,Z 409.781,A -85,B 0,C 180,E1 -6238.752,E2 -6238.752} C_VEL
LIN {X 0,Y 501.215,Z 390.217,A -85,B 0,C 180,E1 -6240.912,E2 -6240.912} C_VEL
LIN {X 0,Y 497.449,Z 375.497,A -85,B 0,C 180,E1 -6242.832,E2 -6242.832} C_VEL
LIN {X 0,Y 495.746,Z 369.359,A -85,B 0,C 180,E1 -6243.686,E2 -6243.686} C_VEL
LIN {X 0,Y 495.679,Z 369.362,A -85,B 0,C 180,E1 -6246.547,E2 -6246.547} C_VEL
LIN {X 0,Y 495.733,Z 369.36,A -85,B 0,C 180,E1 -6249.638,E2 -6249.638} C_VEL
LIN {X 0,Y 495.694,Z 369.361,A -85,B 0,C 180,E1 -6252.885,E2 -6252.885} C_VEL
LIN {X 0,Y 495.702,Z 369.355,A -85,B 0,C 180,E1 -6255.996,E2 -6255.996} C_VEL
LIN {X 0,Y 495.715,Z 369.357,A -85,B 0,C 180,E1 -6259.295,E2 -6259.295} C_VEL
LIN {X 0,Y 495.711,Z 369.356,A -85,B 0,C 180,E1 -6261.405,E2 -6261.405} C_VEL
LIN {X 0,Y 495.715,Z 369.364,A -85,B 0,C 180,E1 -6264.46,E2 -6264.46} C_VEL
LIN {X 0,Y 495.729,Z 369.356,A -85,B 0,C 180,E1 -6267.403,E2 -6267.403} C_VEL
LIN {X 0,Y 495.743,Z 369.36,A -85,B 0,C 180,E1 -6270.252,E2 -6270.252} C_VEL
LIN {X 0,Y 495.724,Z 369.357,A -85,B 0,C 180,E1 -6273.27,E2 -6273.27} C_VEL
LIN {X 0,Y 495.694,Z 369.361,A -85,B 0,C 180,E1 -6275.722,E2 -6275.722} C_VEL
LIN {X 0,Y 495.71,Z 369.365,A -85,B 0,C 180,E1 -6278.37,E2 -6278.37} C_VEL
LIN {X 0,Y 495.734,Z 369.358,A -85,B 0,C 180,E1 -6280.97,E2 -6280.97} C_VEL
LIN {X 0,Y 495.787,Z 369.355,A -85,B 0,C 180,E1 -6284.558,E2 -6284.558} C_VEL
LIN {X 0,Y 495.813,Z 369.348,A -85,B 0,C 180,E1 -6287.966,E2 -6287.966} C_VEL
LIN {X 0,Y 495.781,Z 369.351,A -85,B 0,C 180,E1 -6291.029,E2 -6291.029} C_VEL
LIN {X 0,Y 495.788,Z 369.345,A -85,B 0,C 180,E1 -6293.489,E2 -6293.489} C_VEL
LIN {X 0,Y 495.703,Z 369.36,A -85,B 0,C 180,E1 -6295.935,E2 -6295.935} C_VEL
LIN {X 0,Y 495.963,Z 369.323,A -85,B 0,C 180,E1 -6297.564,E2 -6297.564} C_VEL
LIN {X 0,Y 495.945,Z 369.331,A -85,B 0,C 180,E1 -6300.812,E2 -6300.812} C_VEL
LIN {X 0,Y 495.963,Z 369.33,A -85,B 0,C 180,E1 -6302.437,E2 -6302.437} C_VEL
LIN {X 0,Y 495.86,Z 369.333,A -85,B 0,C 180,E1 -6305.694,E2 -6305.694} C_VEL
LIN {X 0,Y 495.813,Z 369.336,A -85,B 0,C 180,E1 -6308.149,E2 -6308.149} C_VEL
LIN {X 0,Y 495.834,Z 369.342,A -85,B 0,C 180,E1 -6311.446,E2 -6311.446} C_VEL
LIN {X 0,Y 495.766,Z 369.346,A -85,B 0,C 180,E1 -6314.784,E2 -6314.784} C_VEL
LIN {X 0,Y 495.748,Z 369.355,A -85,B 0,C 180,E1 -6317.32,E2 -6317.32} C_VEL
LIN {X 0,Y 495.756,Z 369.347,A -85,B 0,C 180,E1 -6319.891,E2 -6319.891} C_VEL
LIN {X 0,Y 495.745,Z 369.359,A -85,B 0,C 180,E1 -6322.861,E2 -6322.861} C_VEL
LIN {X 0,Y 495.703,Z 369.355,A -85,B 0,C 180,E1 -6326.073,E2 -6326.073} C_VEL
LIN {X 0,Y 495.722,Z 369.363,A -85,B 0,C 180,E1 -6328.818,E2 -6328.818} C_VEL
LIN {X 0,Y 495.743,Z 369.348,A -85,B 0,C 180,E1 -6331.726,E2 -6331.726} C_VEL
LIN {X 0,Y 495.752,Z 369.36,A -85,B 0,C 180,E1 -6334.694,E2 -6334.694} C_VEL
LIN {X 0,Y 495.719,Z 369.358,A -85,B 0,C 180,E1 -6337.563,E2 -6337.563} C_VEL
LIN {X 0,Y 495.735,Z 369.354,A -85,B 0,C 180,E1 -6340.046,E2 -6340.046} C_VEL
LIN {X 0,Y 495.696,Z 369.367,A -85,B 0,C 180,E1 -6342.887,E2 -6342.887} C_VEL
LIN {X 0,Y 495.717,Z 369.358,A -85,B 0,C 180,E1 -6345.999,E2 -6345.999} C_VEL
LIN {X 0,Y 495.725,Z 369.359,A -85,B 0,C 180,E1 -6349.298,E2 -6349.298} C_VEL
LIN {X 0,Y 495.74,Z 369.356,A -85,B 0,C 180,E1 -6351.409,E2 -6351.409} C_VEL
LIN {X 0,Y 495.738,Z 369.355,A -85,B 0,C 180,E1 -6354.463,E2 -6354.463} C_VEL
LIN {X 0,Y 495.747,Z 369.359,A -85,B 0,C 180,E1 -6357.405,E2 -6357.405} C_VEL
LIN {X 0,Y 495.758,Z 369.356,A -85,B 0,C 180,E1 -6358.671,E2 -6358.671} C_VEL
LIN {X 0,Y 496.917,Z 372.469,A -85,B 0,C 180,E1 -6358.79,E2 -6358.79} C_VEL
LIN {X 0,Y 502.159,Z 384.325,A -85,B 0,C 180,E1 -6359.24,E2 -6359.24} C_VEL
LIN {X 0,Y 502.126,Z 391.852,A -85,B 0,C 180,E1 -6359.354,E2 -6359.354} C_VEL
LIN {X 0,Y 501.428,Z 397.708,A -85,B 0,C 180,E1 -6359.409,E2 -6359.409} C_VEL
LIN {X 0,Y 495.925,Z 416.784,A -85,B 0,C 180,E1 -6359.428,E2 -6359.428} C_VEL
LIN {X 0,Y 495.277,Z 422.636,A -85,B 0,C 180,E1 -6359.486,E2 -6359.486} C_VEL
LIN {X 0,Y 494.619,Z 498.692,A -85,B 0,C 180,E1 -6360.647,E2 -6360.647} C_VEL
LIN {X 0,Y 494.411,Z 513.909,A -85,B 0,C 180,E1 -6361.027,E2 -6361.027} C_VEL
LIN {X 0,Y 494.06,Z 528.121,A -85,B 0,C 180,E1 -6361.542,E2 -6361.542} C_VEL
LIN {X 0,Y 493.587,Z 542.254,A -85,B 0,C 180,E1 -6362.222,E2 -6362.222} C_VEL
LIN {X 0,Y 493.064,Z 554.753,A -85,B 0,C 180,E1 -6362.979,E2 -6362.979} C_VEL
LIN {X 0,Y 492.423,Z 567.359,A -85,B 0,C 180,E1 -6363.908,E2 -6363.908} C_VEL
LIN {X 0,Y 491.757,Z 579.1,A -85,B 0,C 180,E1 -6364.952,E2 -6364.952} C_VEL
LIN {X 0,Y 491.097,Z 590.552,A -85,B 0,C 180,E1 -6366.178,E2 -6366.178} C_VEL
LIN {X 0,Y 490.452,Z 600.635,A -85,B 0,C 180,E1 -6367.462,E2 -6367.462} C_VEL
LIN {X 0,Y 489.975,Z 609.436,A -85,B 0,C 180,E1 -6368.802,E2 -6368.802} C_VEL
LIN {X 0,Y 489.414,Z 617.572,A -85,B 0,C 180,E1 -6370.279,E2 -6370.279} C_VEL
LIN {X 0,Y 489.13,Z 623.512,A -85,B 0,C 180,E1 -6371.573,E2 -6371.573} C_VEL
LIN {X 0,Y 488.769,Z 629.972,A -85,B 0,C 180,E1 -6373.288,E2 -6373.288} C_VEL
LIN {X 0,Y 488.567,Z 634.926,A -85,B 0,C 180,E1 -6374.994,E2 -6374.994} C_VEL
LIN {X 0,Y 488.365,Z 638.547,A -85,B 0,C 180,E1 -6376.689,E2 -6376.689} C_VEL
LIN {X 0,Y 488.327,Z 640.934,A -85,B 0,C 180,E1 -6378.377,E2 -6378.377} C_VEL
LIN {X 0,Y 488.261,Z 642.156,A -85,B 0,C 180,E1 -6380.054,E2 -6380.054} C_VEL
LIN {X 0,Y 488.27,Z 642.218,A -85,B 0,C 180,E1 -6381.725,E2 -6381.725} C_VEL
LIN {X 0,Y 488.339,Z 641.184,A -85,B 0,C 180,E1 -6383.389,E2 -6383.389} C_VEL
LIN {X 0,Y 488.365,Z 639.062,A -85,B 0,C 180,E1 -6385.047,E2 -6385.047} C_VEL
LIN {X 0,Y 488.575,Z 635.775,A -85,B 0,C 180,E1 -6386.702,E2 -6386.702} C_VEL
LIN {X 0,Y 488.663,Z 631.314,A -85,B 0,C 180,E1 -6388.352,E2 -6388.352} C_VEL
LIN {X 0,Y 488.952,Z 625.505,A -85,B 0,C 180,E1 -6390,E2 -6390} C_VEL
LIN {X 0,Y 489.417,Z 618.2,A -85,B 0,C 180,E1 -6391.646,E2 -6391.646} C_VEL
LIN {X 0,Y 489.839,Z 610.412,A -85,B 0,C 180,E1 -6393.084,E2 -6393.084} C_VEL
LIN {X 0,Y 490.426,Z 601.076,A -85,B 0,C 180,E1 -6394.521,E2 -6394.521} C_VEL
LIN {X 0,Y 490.983,Z 591.558,A -85,B 0,C 180,E1 -6395.751,E2 -6395.751} C_VEL
LIN {X 0,Y 491.589,Z 580.286,A -85,B 0,C 180,E1 -6396.98,E2 -6396.98} C_VEL
LIN {X 0,Y 492.287,Z 567.833,A -85,B 0,C 180,E1 -6398.105,E2 -6398.105} C_VEL
LIN {X 0,Y 492.907,Z 555.517,A -85,B 0,C 180,E1 -6399.024,E2 -6399.024} C_VEL
LIN {X 0,Y 493.491,Z 542.098,A -85,B 0,C 180,E1 -6399.84,E2 -6399.84} C_VEL
LIN {X 0,Y 494.006,Z 527.63,A -85,B 0,C 180,E1 -6400.531,E2 -6400.531} C_VEL
LIN {X 0,Y 494.286,Z 512.783,A -85,B 0,C 180,E1 -6401.065,E2 -6401.065} C_VEL
LIN {X 0,Y 494.483,Z 497.984,A -85,B 0,C 180,E1 -6401.428,E2 -6401.428} C_VEL
LIN {X 0,Y 495.4,Z 385.784,A -85,B 0,C 180,E1 -6403.12,E2 -6403.12} C_VEL
LIN {X 0,Y 488.76,Z 370.637,A -85,B 0,C 180,E1 -6403.672,E2 -6403.672} C_VEL
LIN {X 0,Y 488.72,Z 370.233,A -85,B 0,C 180,E1 -6403.726,E2 -6403.726} C_VEL
LIN {X 0,Y 488.682,Z 370.239,A -85,B 0,C 180,E1 -6406.716,E2 -6406.716} C_VEL
LIN {X 0,Y 488.71,Z 370.235,A -85,B 0,C 180,E1 -6409.314,E2 -6409.314} C_VEL
LIN {X 0,Y 488.685,Z 370.234,A -85,B 0,C 180,E1 -6411.957,E2 -6411.957} C_VEL
LIN {X 0,Y 488.69,Z 370.24,A -85,B 0,C 180,E1 -6415.038,E2 -6415.038} C_VEL
LIN {X 0,Y 488.684,Z 370.235,A -85,B 0,C 180,E1 -6418.332,E2 -6418.332} C_VEL
LIN {X 0,Y 488.657,Z 370.24,A -85,B 0,C 180,E1 -6421.182,E2 -6421.182} C_VEL
LIN {X 0,Y 488.707,Z 370.229,A -85,B 0,C 180,E1 -6424.114,E2 -6424.114} C_VEL
LIN {X 0,Y 488.645,Z 370.244,A -85,B 0,C 180,E1 -6427.161,E2 -6427.161} C_VEL
LIN {X 0,Y 488.664,Z 370.233,A -85,B 0,C 180,E1 -6430.329,E2 -6430.329} C_VEL
LIN {X 0,Y 488.66,Z 370.237,A -85,B 0,C 180,E1 -6433.656,E2 -6433.656} C_VEL
LIN {X 0,Y 488.661,Z 370.236,A -85,B 0,C 180,E1 -6436.342,E2 -6436.342} C_VEL
LIN {X 0,Y 488.699,Z 370.234,A -85,B 0,C 180,E1 -6439.673,E2 -6439.673} C_VEL
LIN {X 0,Y 488.651,Z 370.238,A -85,B 0,C 180,E1 -6442.838,E2 -6442.838} C_VEL
LIN {X 0,Y 488.703,Z 370.228,A -85,B 0,C 180,E1 -6445.885,E2 -6445.885} C_VEL
LIN {X 0,Y 488.651,Z 370.24,A -85,B 0,C 180,E1 -6448.817,E2 -6448.817} C_VEL
LIN {X 0,Y 488.677,Z 370.237,A -85,B 0,C 180,E1 -6451.667,E2 -6451.667} C_VEL
LIN {X 0,Y 488.683,Z 370.236,A -85,B 0,C 180,E1 -6454.961,E2 -6454.961} C_VEL
LIN {X 0,Y 488.688,Z 370.234,A -85,B 0,C 180,E1 -6458.042,E2 -6458.042} C_VEL
LIN {X 0,Y 488.721,Z 370.227,A -85,B 0,C 180,E1 -6460.685,E2 -6460.685} C_VEL
LIN {X 0,Y 488.748,Z 370.225,A -85,B 0,C 180,E1 -6464.144,E2 -6464.144} C_VEL
LIN {X 0,Y 488.726,Z 370.22,A -85,B 0,C 180,E1 -6467.543,E2 -6467.543} C_VEL
LIN {X 0,Y 488.728,Z 370.216,A -85,B 0,C 180,E1 -6470.063,E2 -6470.063} C_VEL
LIN {X 0,Y 488.809,Z 370.214,A -85,B 0,C 180,E1 -6472.769,E2 -6472.769} C_VEL
LIN {X 0,Y 488.776,Z 370.224,A -85,B 0,C 180,E1 -6475.051,E2 -6475.051} C_VEL
LIN {X 0,Y 488.927,Z 370.204,A -85,B 0,C 180,E1 -6477.528,E2 -6477.528} C_VEL
LIN {X 0,Y 488.925,Z 370.205,A -85,B 0,C 180,E1 -6480,E2 -6480} C_VEL
LIN {X 0,Y 488.934,Z 370.199,A -85,B 0,C 180,E1 -6482.471,E2 -6482.471} C_VEL
LIN {X 0,Y 488.791,Z 370.225,A -85,B 0,C 180,E1 -6485.776,E2 -6485.776} C_VEL
LIN {X 0,Y 488.747,Z 370.223,A -85,B 0,C 180,E1 -6488.267,E2 -6488.267} C_VEL
LIN {X 0,Y 488.793,Z 370.227,A -85,B 0,C 180,E1 -6491.613,E2 -6491.613} C_VEL
LIN {X 0,Y 488.735,Z 370.224,A -85,B 0,C 180,E1 -6495.001,E2 -6495.001} C_VEL
LIN {X 0,Y 488.696,Z 370.229,A -85,B 0,C 180,E1 -6498.444,E2 -6498.444} C_VEL
LIN {X 0,Y 488.68,Z 370.235,A -85,B 0,C 180,E1 -6501.072,E2 -6501.072} C_VEL
LIN {X 0,Y 488.656,Z 370.243,A -85,B 0,C 180,E1 -6503.747,E2 -6503.747} C_VEL
LIN {X 0,Y 488.672,Z 370.233,A -85,B 0,C 180,E1 -6506.477,E2 -6506.477} C_VEL
LIN {X 0,Y 488.69,Z 370.235,A -85,B 0,C 180,E1 -6509.272,E2 -6509.272} C_VEL
LIN {X 0,Y 488.681,Z 370.235,A -85,B 0,C 180,E1 -6512.149,E2 -6512.149} C_VEL
LIN {X 0,Y 488.697,Z 370.231,A -85,B 0,C 180,E1 -6515.117,E2 -6515.117} C_VEL
LIN {X 0,Y 488.644,Z 370.237,A -85,B 0,C 180,E1 -6518.203,E2 -6518.203} C_VEL
LIN {X 0,Y 488.687,Z 370.236,A -85,B 0,C 180,E1 -6520.341,E2 -6520.341} C_VEL
LIN {X 0,Y 488.657,Z 370.241,A -85,B 0,C 180,E1 -6523.658,E2 -6523.658} C_VEL
LIN {X 0,Y 488.667,Z 370.24,A -85,B 0,C 180,E1 -6526.344,E2 -6526.344} C_VEL
LIN {X 0,Y 488.661,Z 370.229,A -85,B 0,C 180,E1 -6529.67,E2 -6529.67} C_VEL
LIN {X 0,Y 488.642,Z 370.244,A -85,B 0,C 180,E1 -6532.283,E2 -6532.283} C_VEL
LIN {X 0,Y 488.726,Z 370.235,A -85,B 0,C 180,E1 -6535.887,E2 -6535.887} C_VEL
LIN {X 0,Y 488.751,Z 370.379,A -85,B 0,C 180,E1 -6536.216,E2 -6536.216} C_VEL
LIN {X 0,Y 494.22,Z 391.394,A -85,B 0,C 180,E1 -6538.917,E2 -6538.917} C_VEL
LIN {X 0,Y 493.514,Z 412.788,A -85,B 0,C 180,E1 -6541.274,E2 -6541.274} C_VEL
LIN {X 0,Y 492.49,Z 440.828,A -85,B 0,C 180,E1 -6544.313,E2 -6544.313} C_VEL
LIN {X 0,Y 491.682,Z 465.111,A -85,B 0,C 180,E1 -6546.917,E2 -6546.917} C_VEL
LIN {X 0,Y 495.308,Z 490.559,A -85,B 0,C 180,E1 -6547.474,E2 -6547.474} C_VEL
LIN {X 0,Y 493.91,Z 634.471,A -85,B 0,C 180,E1 -6549.625,E2 -6549.625} C_VEL
LIN {X 0,Y 493.373,Z 650.726,A -85,B 0,C 180,E1 -6550.042,E2 -6550.042} C_VEL
LIN {X 0,Y 492.765,Z 665.944,A -85,B 0,C 180,E1 -6550.61,E2 -6550.61} C_VEL
LIN {X 0,Y 492.081,Z 681.124,A -85,B 0,C 180,E1 -6551.364,E2 -6551.364} C_VEL
LIN {X 0,Y 491.41,Z 694.557,A -85,B 0,C 180,E1 -6552.2,E2 -6552.2} C_VEL
LIN {X 0,Y 490.673,Z 708.265,A -85,B 0,C 180,E1 -6553.247,E2 -6553.247} C_VEL
LIN {X 0,Y 489.992,Z 720.785,A -85,B 0,C 180,E1 -6554.399,E2 -6554.399} C_VEL
LIN {X 0,Y 489.445,Z 732.254,A -85,B 0,C 180,E1 -6555.659,E2 -6555.659} C_VEL
LIN {X 0,Y 488.953,Z 743.421,A -85,B 0,C 180,E1 -6557.127,E2 -6557.127} C_VEL
LIN {X 0,Y 488.639,Z 752.749,A -85,B 0,C 180,E1 -6558.594,E2 -6558.594} C_VEL
LIN {X 0,Y 488.321,Z 760.49,A -85,B 0,C 180,E1 -6560.055,E2 -6560.055} C_VEL
LIN {X 0,Y 488.223,Z 767.754,A -85,B 0,C 180,E1 -6561.723,E2 -6561.723} C_VEL
LIN {X 0,Y 488.14,Z 773.598,A -85,B 0,C 180,E1 -6563.427,E2 -6563.427} C_VEL
LIN {X 0,Y 488.087,Z 777.796,A -85,B 0,C 180,E1 -6565.044,E2 -6565.044} C_VEL
LIN {X 0,Y 488.068,Z 780.832,A -85,B 0,C 180,E1 -6566.698,E2 -6566.698} C_VEL
LIN {X 0,Y 488.021,Z 782.633,A -85,B 0,C 180,E1 -6568.349,E2 -6568.349} C_VEL
LIN {X 0,Y 488.042,Z 783.25,A -85,B 0,C 180,E1 -6570,E2 -6570} C_VEL
LIN {X 0,Y 488.023,Z 782.615,A -85,B 0,C 180,E1 -6571.65,E2 -6571.65} C_VEL
LIN {X 0,Y 488.071,Z 780.796,A -85,B 0,C 180,E1 -6573.302,E2 -6573.302} C_VEL
LIN {X 0,Y 488.086,Z 777.748,A -85,B 0,C 180,E1 -6574.956,E2 -6574.956} C_VEL
LIN {X 0,Y 488.137,Z 773.41,A -85,B 0,C 180,E1 -6576.614,E2 -6576.614} C_VEL
LIN {X 0,Y 488.222,Z 767.67,A -85,B 0,C 180,E1 -6578.276,E2 -6578.276} C_VEL
LIN {X 0,Y 488.323,Z 760.375,A -85,B 0,C 180,E1 -6579.945,E2 -6579.945} C_VEL
LIN {X 0,Y 488.63,Z 752.612,A -85,B 0,C 180,E1 -6581.406,E2 -6581.406} C_VEL
LIN {X 0,Y 488.952,Z 743.262,A -85,B 0,C 180,E1 -6582.872,E2 -6582.872} C_VEL
LIN {X 0,Y 489.446,Z 732.064,A -85,B 0,C 180,E1 -6584.34,E2 -6584.34} C_VEL
LIN {X 0,Y 490.062,Z 719.517,A -85,B 0,C 180,E1 -6585.704,E2 -6585.704} C_VEL
LIN {X 0,Y 490.726,Z 706.769,A -85,B 0,C 180,E1 -6586.858,E2 -6586.858} C_VEL
LIN {X 0,Y 491.445,Z 692.712,A -85,B 0,C 180,E1 -6587.906,E2 -6587.906} C_VEL
LIN {X 0,Y 492.101,Z 678.948,A -85,B 0,C 180,E1 -6588.743,E2 -6588.743} C_VEL
LIN {X 0,Y 492.812,Z 663.788,A -85,B 0,C 180,E1 -6589.469,E2 -6589.469} C_VEL
LIN {X 0,Y 493.444,Z 648.543,A -85,B 0,C 180,E1 -6590.014,E2 -6590.014} C_VEL
LIN {X 0,Y 493.897,Z 632.73,A -85,B 0,C 180,E1 -6590.402,E2 -6590.402} C_VEL
LIN {X 0,Y 495.3,Z 490.539,A -85,B 0,C 180,E1 -6592.526,E2 -6592.526} C_VEL
LIN {X 0,Y 491.644,Z 464.452,A -85,B 0,C 180,E1 -6593.12,E2 -6593.12} C_VEL
LIN {X 0,Y 492.844,Z 431.454,A -85,B 0,C 180,E1 -6596.691,E2 -6596.691} C_VEL
LIN {X 0,Y 494.03,Z 401.795,A -85,B 0,C 180,E1 -6599.978,E2 -6599.978} C_VEL
LIN {X 0,Y 494.476,Z 392.038,A -85,B 0,C 180,E1 -6601.077,E2 -6601.077} C_VEL
LIN {X 0,Y 490.318,Z 375.883,A -85,B 0,C 180,E1 -6603.232,E2 -6603.232} C_VEL
LIN {X 0,Y 488.724,Z 370.234,A -85,B 0,C 180,E1 -6604.029,E2 -6604.029} C_VEL
LIN {X 0,Y 488.64,Z 370.24,A -85,B 0,C 180,E1 -6607.161,E2 -6607.161} C_VEL
LIN {X 0,Y 488.685,Z 370.239,A -85,B 0,C 180,E1 -6610.34,E2 -6610.34} C_VEL
LIN {X 0,Y 488.664,Z 370.238,A -85,B 0,C 180,E1 -6613.655,E2 -6613.655} C_VEL
LIN {X 0,Y 488.653,Z 370.236,A -85,B 0,C 180,E1 -6616.342,E2 -6616.342} C_VEL
LIN {X 0,Y 488.693,Z 370.233,A -85,B 0,C 180,E1 -6619.673,E2 -6619.673} C_VEL
LIN {X 0,Y 488.636,Z 370.241,A -85,B 0,C 180,E1 -6622.837,E2 -6622.837} C_VEL
LIN {X 0,Y 488.702,Z 370.236,A -85,B 0,C 180,E1 -6625.885,E2 -6625.885} C_VEL
LIN {X 0,Y 488.667,Z 370.236,A -85,B 0,C 180,E1 -6628.819,E2 -6628.819} C_VEL
LIN {X 0,Y 488.677,Z 370.237,A -85,B 0,C 180,E1 -6631.667,E2 -6631.667} C_VEL
LIN {X 0,Y 488.683,Z 370.234,A -85,B 0,C 180,E1 -6634.959,E2 -6634.959} C_VEL
LIN {X 0,Y 488.667,Z 370.241,A -85,B 0,C 180,E1 -6638.042,E2 -6638.042} C_VEL
LIN {X 0,Y 488.692,Z 370.238,A -85,B 0,C 180,E1 -6640.685,E2 -6640.685} C_VEL
LIN {X 0,Y 488.694,Z 370.237,A -85,B 0,C 180,E1 -6644.143,E2 -6644.143} C_VEL
LIN {X 0,Y 488.691,Z 370.238,A -85,B 0,C 180,E1 -6646.697,E2 -6646.697} C_VEL
LIN {X 0,Y 488.71,Z 370.229,A -85,B 0,C 180,E1 -6649.225,E2 -6649.225} C_VEL
LIN {X 0,Y 488.785,Z 370.225,A -85,B 0,C 180,E1 -6652.565,E2 -6652.565} C_VEL
LIN {X 0,Y 488.767,Z 370.225,A -85,B 0,C 180,E1 -6655.051,E2 -6655.051} C_VEL
LIN {X 0,Y 488.931,Z 370.199,A -85,B 0,C 180,E1 -6657.529,E2 -6657.529} C_VEL
LIN {X 0,Y 488.897,Z 370.209,A -85,B 0,C 180,E1 -6660.824,E2 -6660.824} C_VEL
LIN {X 0,Y 488.93,Z 370.207,A -85,B 0,C 180,E1 -6662.472,E2 -6662.472} C_VEL
LIN {X 0,Y 488.818,Z 370.21,A -85,B 0,C 180,E1 -6665.776,E2 -6665.776} C_VEL
LIN {X 0,Y 488.759,Z 370.215,A -85,B 0,C 180,E1 -6668.268,E2 -6668.268} C_VEL
LIN {X 0,Y 488.789,Z 370.219,A -85,B 0,C 180,E1 -6671.613,E2 -6671.613} C_VEL
LIN {X 0,Y 488.742,Z 370.223,A -85,B 0,C 180,E1 -6675.001,E2 -6675.001} C_VEL
LIN {X 0,Y 488.734,Z 370.231,A -85,B 0,C 180,E1 -6678.443,E2 -6678.443} C_VEL
LIN {X 0,Y 488.694,Z 370.227,A -85,B 0,C 180,E1 -6681.072,E2 -6681.072} C_VEL
LIN {X 0,Y 488.656,Z 370.237,A -85,B 0,C 180,E1 -6683.748,E2 -6683.748} C_VEL
LIN {X 0,Y 488.686,Z 370.231,A -85,B 0,C 180,E1 -6686.923,E2 -6686.923} C_VEL
LIN {X 0,Y 488.711,Z 370.233,A -85,B 0,C 180,E1 -6690.22,E2 -6690.22} C_VEL
LIN {X 0,Y 488.701,Z 370.234,A -85,B 0,C 180,E1 -6693.481,E2 -6693.481} C_VEL
LIN {X 0,Y 488.672,Z 370.235,A -85,B 0,C 180,E1 -6696.355,E2 -6696.355} C_VEL
LIN {X 0,Y 488.684,Z 370.236,A -85,B 0,C 180,E1 -6699.256,E2 -6699.256} C_VEL
LIN {X 0,Y 488.659,Z 370.24,A -85,B 0,C 180,E1 -6702.529,E2 -6702.529} C_VEL
LIN {X 0,Y 488.694,Z 370.239,A -85,B 0,C 180,E1 -6705.198,E2 -6705.198} C_VEL
LIN {X 0,Y 488.67,Z 370.239,A -85,B 0,C 180,E1 -6708.582,E2 -6708.582} C_VEL
LIN {X 0,Y 488.693,Z 370.24,A -85,B 0,C 180,E1 -6710.95,E2 -6710.95} C_VEL
LIN {X 0,Y 488.664,Z 370.235,A -85,B 0,C 180,E1 -6713.868,E2 -6713.868} C_VEL
LIN {X 0,Y 488.698,Z 370.238,A -85,B 0,C 180,E1 -6716.875,E2 -6716.875} C_VEL
LIN {X 0,Y 488.702,Z 370.233,A -85,B 0,C 180,E1 -6718.306,E2 -6718.306} C_VEL
LIN {X 0,Y 489.819,Z 373.225,A -85,B 0,C 180,E1 -6718.425,E2 -6718.425} C_VEL
LIN {X 0,Y 495.721,Z 386.624,A -85,B 0,C 180,E1 -6718.948,E2 -6718.948} C_VEL
LIN {X 0,Y 495.277,Z 422.636,A -85,B 0,C 180,E1 -6719.486,E2 -6719.486} C_VEL
LIN {X 0,Y 494.617,Z 426.562,A -85,B 0,C 180,E1 -6719.514,E2 -6719.514} C_VEL
LIN {X 0,Y 489.18,Z 438.921,A -85,B 0,C 180,E1 -6719.43,E2 -6719.43} C_VEL
LIN {X 0,Y 488.551,Z 442.844,A -85,B 0,C 180,E1 -6719.46,E2 -6719.46} C_VEL
LIN {X 0,Y 488.066,Z 500.607,A -85,B 0,C 180,E1 -6720.363,E2 -6720.363} C_VEL
LIN {X 0,Y 487.809,Z 515.899,A -85,B 0,C 180,E1 -6720.759,E2 -6720.759} C_VEL
LIN {X 0,Y 487.422,Z 530.145,A -85,B 0,C 180,E1 -6721.295,E2 -6721.295} C_VEL
LIN {X 0,Y 486.94,Z 544.2,A -85,B 0,C 180,E1 -6721.994,E2 -6721.994} C_VEL
LIN {X 0,Y 486.339,Z 557.187,A -85,B 0,C 180,E1 -6722.807,E2 -6722.807} C_VEL
LIN {X 0,Y 485.662,Z 570.029,A -85,B 0,C 180,E1 -6723.793,E2 -6723.793} C_VEL
LIN {X 0,Y 484.935,Z 582.133,A -85,B 0,C 180,E1 -6724.919,E2 -6724.919} C_VEL
LIN {X 0,Y 484.257,Z 592.824,A -85,B 0,C 180,E1 -6726.11,E2 -6726.11} C_VEL
LIN {X 0,Y 483.604,Z 602.276,A -85,B 0,C 180,E1 -6727.35,E2 -6727.35} C_VEL
LIN {X 0,Y 483.09,Z 610.789,A -85,B 0,C 180,E1 -6728.673,E2 -6728.673} C_VEL
LIN {X 0,Y 482.493,Z 619.038,A -85,B 0,C 180,E1 -6730.206,E2 -6730.206} C_VEL
LIN {X 0,Y 482.147,Z 625.821,A -85,B 0,C 180,E1 -6731.746,E2 -6731.746} C_VEL
LIN {X 0,Y 481.766,Z 631.966,A -85,B 0,C 180,E1 -6733.474,E2 -6733.474} C_VEL
LIN {X 0,Y 481.546,Z 636.667,A -85,B 0,C 180,E1 -6735.203,E2 -6735.203} C_VEL
LIN {X 0,Y 481.387,Z 639.349,A -85,B 0,C 180,E1 -6736.492,E2 -6736.492} C_VEL
LIN {X 0,Y 481.299,Z 641.821,A -85,B 0,C 180,E1 -6738.204,E2 -6738.204} C_VEL
LIN {X 0,Y 481.254,Z 643.098,A -85,B 0,C 180,E1 -6739.908,E2 -6739.908} C_VEL
LIN {X 0,Y 481.259,Z 643.255,A -85,B 0,C 180,E1 -6741.603,E2 -6741.603} C_VEL
LIN {X 0,Y 481.31,Z 642.316,A -85,B 0,C 180,E1 -6743.292,E2 -6743.292} C_VEL
LIN {X 0,Y 481.356,Z 640.286,A -85,B 0,C 180,E1 -6744.975,E2 -6744.975} C_VEL
LIN {X 0,Y 481.57,Z 637.096,A -85,B 0,C 180,E1 -6746.654,E2 -6746.654} C_VEL
LIN {X 0,Y 481.676,Z 632.703,A -85,B 0,C 180,E1 -6748.328,E2 -6748.328} C_VEL
LIN {X 0,Y 481.985,Z 626.981,A -85,B 0,C 180,E1 -6750,E2 -6750} C_VEL
LIN {X 0,Y 482.474,Z 619.791,A -85,B 0,C 180,E1 -6751.67,E2 -6751.67} C_VEL
LIN {X 0,Y 482.977,Z 610.945,A -85,B 0,C 180,E1 -6753.337,E2 -6753.337} C_VEL
LIN {X 0,Y 483.651,Z 601.492,A -85,B 0,C 180,E1 -6754.793,E2 -6754.793} C_VEL
LIN {X 0,Y 484.338,Z 590.127,A -85,B 0,C 180,E1 -6756.248,E2 -6756.248} C_VEL
LIN {X 0,Y 484.996,Z 578.346,A -85,B 0,C 180,E1 -6757.494,E2 -6757.494} C_VEL
LIN {X 0,Y 485.761,Z 565.219,A -85,B 0,C 180,E1 -6758.633,E2 -6758.633} C_VEL
LIN {X 0,Y 486.462,Z 552.101,A -85,B 0,C 180,E1 -6759.564,E2 -6759.564} C_VEL
LIN {X 0,Y 487.02,Z 538.552,A -85,B 0,C 180,E1 -6760.34,E2 -6760.34} C_VEL
LIN {X 0,Y 487.526,Z 523.384,A -85,B 0,C 180,E1 -6761.008,E2 -6761.008} C_VEL
LIN {X 0,Y 487.758,Z 508.654,A -85,B 0,C 180,E1 -6761.485,E2 -6761.485} C_VEL
LIN {X 0,Y 487.893,Z 494.091,A -85,B 0,C 180,E1 -6761.793,E2 -6761.793} C_VEL
LIN {X 0,Y 488.801,Z 387.633,A -85,B 0,C 180,E1 -6763.405,E2 -6763.405} C_VEL
LIN {X 0,Y 481.714,Z 371.497,A -85,B 0,C 180,E1 -6764.004,E2 -6764.004} C_VEL
LIN {X 0,Y 481.654,Z 371.113,A -85,B 0,C 180,E1 -6764.023,E2 -6764.023} C_VEL
LIN {X 0,Y 481.647,Z 371.112,A -85,B 0,C 180,E1 -6766.095,E2 -6766.095} C_VEL
LIN {X 0,Y 481.652,Z 371.115,A -85,B 0,C 180,E1 -6768.724,E2 -6768.724} C_VEL
LIN {X 0,Y 481.636,Z 371.116,A -85,B 0,C 180,E1 -6771.395,E2 -6771.395} C_VEL
LIN {X 0,Y 481.615,Z 371.115,A -85,B 0,C 180,E1 -6774.116,E2 -6774.116} C_VEL
LIN {X 0,Y 481.642,Z 371.118,A -85,B 0,C 180,E1 -6777.114,E2 -6777.114} C_VEL
LIN {X 0,Y 481.599,Z 371.109,A -85,B 0,C 180,E1 -6779.746,E2 -6779.746} C_VEL
LIN {X 0,Y 481.632,Z 371.116,A -85,B 0,C 180,E1 -6782.677,E2 -6782.677} C_VEL
LIN {X 0,Y 481.646,Z 371.118,A -85,B 0,C 180,E1 -6785.201,E2 -6785.201} C_VEL
LIN {X 0,Y 481.624,Z 371.113,A -85,B 0,C 180,E1 -6788.002,E2 -6788.002} C_VEL
LIN {X 0,Y 481.609,Z 371.118,A -85,B 0,C 180,E1 -6791.046,E2 -6791.046} C_VEL
LIN {X 0,Y 481.628,Z 371.111,A -85,B 0,C 180,E1 -6794.46,E2 -6794.46} C_VEL
LIN {X 0,Y 481.608,Z 371.118,A -85,B 0,C 180,E1 -6796.855,E2 -6796.855} C_VEL
LIN {X 0,Y 481.649,Z 371.11,A -85,B 0,C 180,E1 -6800.057,E2 -6800.057} C_VEL
LIN {X 0,Y 481.61,Z 371.122,A -85,B 0,C 180,E1 -6803.378,E2 -6803.378} C_VEL
LIN {X 0,Y 481.665,Z 371.104,A -85,B 0,C 180,E1 -6806.326,E2 -6806.326} C_VEL
LIN {X 0,Y 481.604,Z 371.12,A -85,B 0,C 180,E1 -6809.425,E2 -6809.425} C_VEL
LIN {X 0,Y 481.634,Z 371.111,A -85,B 0,C 180,E1 -6812.164,E2 -6812.164} C_VEL
LIN {X 0,Y 481.657,Z 371.112,A -85,B 0,C 180,E1 -6814.966,E2 -6814.966} C_VEL
LIN {X 0,Y 481.639,Z 371.115,A -85,B 0,C 180,E1 -6817.704,E2 -6817.704} C_VEL
LIN {X 0,Y 481.687,Z 371.102,A -85,B 0,C 180,E1 -6820.392,E2 -6820.392} C_VEL
LIN {X 0,Y 481.656,Z 371.11,A -85,B 0,C 180,E1 -6823.032,E2 -6823.032} C_VEL
LIN {X 0,Y 481.662,Z 371.108,A -85,B 0,C 180,E1 -6825.638,E2 -6825.638} C_VEL
LIN {X 0,Y 481.74,Z 371.082,A -85,B 0,C 180,E1 -6828.215,E2 -6828.215} C_VEL
LIN {X 0,Y 481.702,Z 371.101,A -85,B 0,C 180,E1 -6831.61,E2 -6831.61} C_VEL
LIN {X 0,Y 481.763,Z 371.096,A -85,B 0,C 180,E1 -6834.139,E2 -6834.139} C_VEL
LIN {X 0,Y 481.892,Z 371.08,A -85,B 0,C 180,E1 -6837.492,E2 -6837.492} C_VEL
LIN {X 0,Y 481.895,Z 371.081,A -85,B 0,C 180,E1 -6840,E2 -6840} C_VEL
LIN {X 0,Y 481.901,Z 371.075,A -85,B 0,C 180,E1 -6842.507,E2 -6842.507} C_VEL
LIN {X 0,Y 481.752,Z 371.101,A -85,B 0,C 180,E1 -6845.861,E2 -6845.861} C_VEL
LIN {X 0,Y 481.706,Z 371.099,A -85,B 0,C 180,E1 -6848.389,E2 -6848.389} C_VEL
LIN {X 0,Y 481.74,Z 371.104,A -85,B 0,C 180,E1 -6851.785,E2 -6851.785} C_VEL
LIN {X 0,Y 481.718,Z 371.1,A -85,B 0,C 180,E1 -6855.225,E2 -6855.225} C_VEL
LIN {X 0,Y 481.639,Z 371.107,A -85,B 0,C 180,E1 -6858.724,E2 -6858.724} C_VEL
LIN {X 0,Y 481.619,Z 371.118,A -85,B 0,C 180,E1 -6861.396,E2 -6861.396} C_VEL
LIN {X 0,Y 481.636,Z 371.114,A -85,B 0,C 180,E1 -6864.115,E2 -6864.115} C_VEL
LIN {X 0,Y 481.642,Z 371.11,A -85,B 0,C 180,E1 -6867.117,E2 -6867.117} C_VEL
LIN {X 0,Y 481.655,Z 371.115,A -85,B 0,C 180,E1 -6869.743,E2 -6869.743} C_VEL
LIN {X 0,Y 481.639,Z 371.108,A -85,B 0,C 180,E1 -6872.677,E2 -6872.677} C_VEL
LIN {X 0,Y 481.641,Z 371.111,A -85,B 0,C 180,E1 -6875.202,E2 -6875.202} C_VEL
LIN {X 0,Y 481.619,Z 371.113,A -85,B 0,C 180,E1 -6878.003,E2 -6878.003} C_VEL
LIN {X 0,Y 481.616,Z 371.115,A -85,B 0,C 180,E1 -6881.046,E2 -6881.046} C_VEL
LIN {X 0,Y 481.644,Z 371.112,A -85,B 0,C 180,E1 -6884.459,E2 -6884.459} C_VEL
LIN {X 0,Y 481.609,Z 371.117,A -85,B 0,C 180,E1 -6886.856,E2 -6886.856} C_VEL
LIN {X 0,Y 481.624,Z 371.107,A -85,B 0,C 180,E1 -6890.055,E2 -6890.055} C_VEL
LIN {X 0,Y 481.6,Z 371.119,A -85,B 0,C 180,E1 -6893.252,E2 -6893.252} C_VEL
LIN {X 0,Y 481.709,Z 371.288,A -85,B 0,C 180,E1 -6895.92,E2 -6895.92} C_VEL
LIN {X 0,Y 487.332,Z 392.743,A -85,B 0,C 180,E1 -6898.724,E2 -6898.724} C_VEL
LIN {X 0,Y 487.301,Z 398.015,A -85,B 0,C 180,E1 -6899.324,E2 -6899.324} C_VEL
LIN {X 0,Y 486.369,Z 420.479,A -85,B 0,C 180,E1 -6901.817,E2 -6901.817} C_VEL
LIN {X 0,Y 485.513,Z 443.811,A -85,B 0,C 180,E1 -6904.377,E2 -6904.377} C_VEL
LIN {X 0,Y 484.819,Z 464.34,A -85,B 0,C 180,E1 -6906.587,E2 -6906.587} C_VEL
LIN {X 0,Y 488.694,Z 491.057,A -85,B 0,C 180,E1 -6907.182,E2 -6907.182} C_VEL
LIN {X 0,Y 487.231,Z 633.347,A -85,B 0,C 180,E1 -6909.333,E2 -6909.333} C_VEL
LIN {X 0,Y 486.699,Z 649.437,A -85,B 0,C 180,E1 -6909.749,E2 -6909.749} C_VEL
LIN {X 0,Y 486.045,Z 663.929,A -85,B 0,C 180,E1 -6910.286,E2 -6910.286} C_VEL
LIN {X 0,Y 485.388,Z 678.23,A -85,B 0,C 180,E1 -6910.987,E2 -6910.987} C_VEL
LIN {X 0,Y 484.671,Z 691.973,A -85,B 0,C 180,E1 -6911.835,E2 -6911.835} C_VEL
LIN {X 0,Y 483.854,Z 705.982,A -85,B 0,C 180,E1 -6912.895,E2 -6912.895} C_VEL
LIN {X 0,Y 483.123,Z 718.703,A -85,B 0,C 180,E1 -6914.063,E2 -6914.063} C_VEL
LIN {X 0,Y 482.441,Z 731.223,A -85,B 0,C 180,E1 -6915.446,E2 -6915.446} C_VEL
LIN {X 0,Y 481.94,Z 742.396,A -85,B 0,C 180,E1 -6916.936,E2 -6916.936} C_VEL
LIN {X 0,Y 481.542,Z 751.717,A -85,B 0,C 180,E1 -6918.423,E2 -6918.423} C_VEL
LIN {X 0,Y 481.273,Z 759.468,A -85,B 0,C 180,E1 -6919.908,E2 -6919.908} C_VEL
LIN {X 0,Y 481.167,Z 766.734,A -85,B 0,C 180,E1 -6921.601,E2 -6921.601} C_VEL
LIN {X 0,Y 481.071,Z 772.861,A -85,B 0,C 180,E1 -6923.421,E2 -6923.421} C_VEL
LIN {X 0,Y 481.059,Z 776.784,A -85,B 0,C 180,E1 -6924.971,E2 -6924.971} C_VEL
LIN {X 0,Y 481.029,Z 779.818,A -85,B 0,C 180,E1 -6926.649,E2 -6926.649} C_VEL
LIN {X 0,Y 480.99,Z 781.621,A -85,B 0,C 180,E1 -6928.325,E2 -6928.325} C_VEL
LIN {X 0,Y 481.032,Z 782.238,A -85,B 0,C 180,E1 -6930,E2 -6930} C_VEL
LIN {X 0,Y 480.993,Z 781.597,A -85,B 0,C 180,E1 -6931.674,E2 -6931.674} C_VEL
LIN {X 0,Y 481.033,Z 779.773,A -85,B 0,C 180,E1 -6933.35,E2 -6933.35} C_VEL
LIN {X 0,Y 481.06,Z 776.721,A -85,B 0,C 180,E1 -6935.028,E2 -6935.028} C_VEL
LIN {X 0,Y 481.076,Z 772.372,A -85,B 0,C 180,E1 -6936.711,E2 -6936.711} C_VEL
LIN {X 0,Y 481.167,Z 766.626,A -85,B 0,C 180,E1 -6938.398,E2 -6938.398} C_VEL
LIN {X 0,Y 481.274,Z 759.324,A -85,B 0,C 180,E1 -6940.092,E2 -6940.092} C_VEL
LIN {X 0,Y 481.536,Z 752.72,A -85,B 0,C 180,E1 -6941.363,E2 -6941.363} C_VEL
LIN {X 0,Y 481.863,Z 743.602,A -85,B 0,C 180,E1 -6942.851,E2 -6942.851} C_VEL
LIN {X 0,Y 482.34,Z 732.679,A -85,B 0,C 180,E1 -6944.341,E2 -6944.341} C_VEL
LIN {X 0,Y 482.89,Z 721.501,A -85,B 0,C 180,E1 -6945.619,E2 -6945.619} C_VEL
LIN {X 0,Y 483.621,Z 709.26,A -85,B 0,C 180,E1 -6946.796,E2 -6946.796} C_VEL
LIN {X 0,Y 484.331,Z 696.114,A -85,B 0,C 180,E1 -6947.85,E2 -6947.85} C_VEL
LIN {X 0,Y 485.125,Z 681.548,A -85,B 0,C 180,E1 -6948.803,E2 -6948.803} C_VEL
LIN {X 0,Y 485.89,Z 666.62,A -85,B 0,C 180,E1 -6949.577,E2 -6949.577} C_VEL
LIN {X 0,Y 486.57,Z 651.939,A -85,B 0,C 180,E1 -6950.158,E2 -6950.158} C_VEL
LIN {X 0,Y 487.154,Z 636.682,A -85,B 0,C 180,E1 -6950.587,E2 -6950.587} C_VEL
LIN {X 0,Y 487.445,Z 617.014,A -85,B 0,C 180,E1 -6950.933,E2 -6950.933} C_VEL
LIN {X 0,Y 488.734,Z 491.085,A -85,B 0,C 180,E1 -6952.83,E2 -6952.83} C_VEL
LIN {X 0,Y 484.769,Z 463.458,A -85,B 0,C 180,E1 -6953.467,E2 -6953.467} C_VEL
LIN {X 0,Y 485.998,Z 432.623,A -85,B 0,C 180,E1 -6956.865,E2 -6956.865} C_VEL
LIN {X 0,Y 487.301,Z 403.107,A -85,B 0,C 180,E1 -6960.189,E2 -6960.189} C_VEL
LIN {X 0,Y 487.735,Z 393.883,A -85,B 0,C 180,E1 -6961.247,E2 -6961.247} C_VEL
LIN {X 0,Y 483.835,Z 378.687,A -85,B 0,C 180,E1 -6963.31,E2 -6963.31} C_VEL
LIN {X 0,Y 481.668,Z 371.112,A -85,B 0,C 180,E1 -6964.396,E2 -6964.396} C_VEL
LIN {X 0,Y 481.622,Z 371.119,A -85,B 0,C 180,E1 -6968.002,E2 -6968.002} C_VEL
LIN {X 0,Y 481.617,Z 371.114,A -85,B 0,C 180,E1 -6971.044,E2 -6971.044} C_VEL
LIN {X 0,Y 481.643,Z 371.108,A -85,B 0,C 180,E1 -6974.457,E2 -6974.457} C_VEL
LIN {X 0,Y 481.603,Z 371.119,A -85,B 0,C 180,E1 -6977.835,E2 -6977.835} C_VEL
LIN {X 0,Y 481.636,Z 371.111,A -85,B 0,C 180,E1 -6980.655,E2 -6980.655} C_VEL
LIN {X 0,Y 481.594,Z 371.116,A -85,B 0,C 180,E1 -6983.379,E2 -6983.379} C_VEL
LIN {X 0,Y 481.658,Z 371.113,A -85,B 0,C 180,E1 -6986.326,E2 -6986.326} C_VEL
LIN {X 0,Y 481.627,Z 371.111,A -85,B 0,C 180,E1 -6989.419,E2 -6989.419} C_VEL
LIN {X 0,Y 481.633,Z 371.118,A -85,B 0,C 180,E1 -6992.164,E2 -6992.164} C_VEL
LIN {X 0,Y 481.658,Z 371.109,A -85,B 0,C 180,E1 -6994.967,E2 -6994.967} C_VEL
LIN {X 0,Y 481.618,Z 371.116,A -85,B 0,C 180,E1 -6997.703,E2 -6997.703} C_VEL
LIN {X 0,Y 481.638,Z 371.119,A -85,B 0,C 180,E1 -7000.39,E2 -7000.39} C_VEL
LIN {X 0,Y 481.602,Z 371.117,A -85,B 0,C 180,E1 -7003.031,E2 -7003.031} C_VEL
LIN {X 0,Y 481.65,Z 371.109,A -85,B 0,C 180,E1 -7005.638,E2 -7005.638} C_VEL
LIN {X 0,Y 481.734,Z 371.104,A -85,B 0,C 180,E1 -7008.215,E2 -7008.215} C_VEL
LIN {X 0,Y 481.701,Z 371.103,A -85,B 0,C 180,E1 -7011.611,E2 -7011.611} C_VEL
LIN {X 0,Y 481.749,Z 371.097,A -85,B 0,C 180,E1 -7014.139,E2 -7014.139} C_VEL
LIN {X 0,Y 481.898,Z 371.075,A -85,B 0,C 180,E1 -7017.493,E2 -7017.493} C_VEL
LIN {X 0,Y 481.849,Z 371.086,A -85,B 0,C 180,E1 -7020.836,E2 -7020.836} C_VEL
LIN {X 0,Y 481.896,Z 371.083,A -85,B 0,C 180,E1 -7022.508,E2 -7022.508} C_VEL
LIN {X 0,Y 481.779,Z 371.087,A -85,B 0,C 180,E1 -7025.861,E2 -7025.861} C_VEL
LIN {X 0,Y 481.714,Z 371.094,A -85,B 0,C 180,E1 -7028.389,E2 -7028.389} C_VEL
LIN {X 0,Y 481.735,Z 371.098,A -85,B 0,C 180,E1 -7031.786,E2 -7031.786} C_VEL
LIN {X 0,Y 481.725,Z 371.097,A -85,B 0,C 180,E1 -7035.225,E2 -7035.225} C_VEL
LIN {X 0,Y 481.695,Z 371.108,A -85,B 0,C 180,E1 -7038.723,E2 -7038.723} C_VEL
LIN {X 0,Y 481.632,Z 371.106,A -85,B 0,C 180,E1 -7041.396,E2 -7041.396} C_VEL
LIN {X 0,Y 481.635,Z 371.113,A -85,B 0,C 180,E1 -7044.116,E2 -7044.116} C_VEL
LIN {X 0,Y 481.641,Z 371.109,A -85,B 0,C 180,E1 -7047.118,E2 -7047.118} C_VEL
LIN {X 0,Y 481.659,Z 371.11,A -85,B 0,C 180,E1 -7049.743,E2 -7049.743} C_VEL
LIN {X 0,Y 481.642,Z 371.109,A -85,B 0,C 180,E1 -7052.677,E2 -7052.677} C_VEL
LIN {X 0,Y 481.626,Z 371.112,A -85,B 0,C 180,E1 -7055.711,E2 -7055.711} C_VEL
LIN {X 0,Y 481.657,Z 371.117,A -85,B 0,C 180,E1 -7058.861,E2 -7058.861} C_VEL
LIN {X 0,Y 481.617,Z 371.115,A -85,B 0,C 180,E1 -7062.164,E2 -7062.164} C_VEL
LIN {X 0,Y 481.647,Z 371.112,A -85,B 0,C 180,E1 -7065.543,E2 -7065.543} C_VEL
LIN {X 0,Y 481.625,Z 371.118,A -85,B 0,C 180,E1 -7068.957,E2 -7068.957} C_VEL
LIN {X 0,Y 481.643,Z 371.109,A -85,B 0,C 180,E1 -7071.995,E2 -7071.995} C_VEL
LIN {X 0,Y 481.677,Z 371.113,A -85,B 0,C 180,E1 -7075.318,E2 -7075.318} C_VEL
LIN {X 0,Y 481.653,Z 371.112,A -85,B 0,C 180,E1 -7077.924,E2 -7077.924} C_VEL
LIN {X 0,Y 482.817,Z 374.215,A -85,B 0,C 180,E1 -7078.054,E2 -7078.054} C_VEL
LIN {X 0,Y 489.121,Z 387.968,A -85,B 0,C 180,E1 -7078.622,E2 -7078.622} C_VEL
LIN {X 0,Y 488.551,Z 442.844,A -85,B 0,C 180,E1 -7079.46,E2 -7079.46} C_VEL
LIN {X 0,Y 487.937,Z 448.694,A -85,B 0,C 180,E1 -7079.52,E2 -7079.52} C_VEL
LIN {X 0,Y 482.414,Z 467.763,A -85,B 0,C 180,E1 -7079.535,E2 -7079.535} C_VEL
LIN {X 0,Y 481.746,Z 473.617,A -85,B 0,C 180,E1 -7079.594,E2 -7079.594} C_VEL
LIN {X 0,Y 481.52,Z 503.597,A -85,B 0,C 180,E1 -7080.092,E2 -7080.092} C_VEL
LIN {X 0,Y 481.2,Z 519.224,A -85,B 0,C 180,E1 -7080.528,E2 -7080.528} C_VEL
LIN {X 0,Y 480.84,Z 533.55,A -85,B 0,C 180,E1 -7081.104,E2 -7081.104} C_VEL
LIN {X 0,Y 480.167,Z 548.572,A -85,B 0,C 180,E1 -7081.898,E2 -7081.898} C_VEL
LIN {X 0,Y 479.548,Z 561.271,A -85,B 0,C 180,E1 -7082.744,E2 -7082.744} C_VEL
LIN {X 0,Y 478.844,Z 573.951,A -85,B 0,C 180,E1 -7083.779,E2 -7083.779} C_VEL
LIN {X 0,Y 478.053,Z 586.27,A -85,B 0,C 180,E1 -7084.998,E2 -7084.998} C_VEL
LIN {X 0,Y 477.329,Z 596.765,A -85,B 0,C 180,E1 -7086.244,E2 -7086.244} C_VEL
LIN {X 0,Y 476.533,Z 606.933,A -85,B 0,C 180,E1 -7087.682,E2 -7087.682} C_VEL
LIN {X 0,Y 475.924,Z 616.049,A -85,B 0,C 180,E1 -7089.244,E2 -7089.244} C_VEL
LIN {X 0,Y 475.447,Z 622.526,A -85,B 0,C 180,E1 -7090.575,E2 -7090.575} C_VEL
LIN {X 0,Y 475.019,Z 629.627,A -85,B 0,C 180,E1 -7092.345,E2 -7092.345} C_VEL
LIN {X 0,Y 474.669,Z 635.524,A -85,B 0,C 180,E1 -7094.239,E2 -7094.239} C_VEL
LIN {X 0,Y 474.518,Z 638.406,A -85,B 0,C 180,E1 -7095.418,E2 -7095.418} C_VEL
LIN {X 0,Y 474.296,Z 641.566,A -85,B 0,C 180,E1 -7097.158,E2 -7097.158} C_VEL
LIN {X 0,Y 474.251,Z 643.503,A -85,B 0,C 180,E1 -7098.893,E2 -7098.893} C_VEL
LIN {X 0,Y 474.225,Z 644.308,A -85,B 0,C 180,E1 -7100.618,E2 -7100.618} C_VEL
LIN {X 0,Y 474.271,Z 644.003,A -85,B 0,C 180,E1 -7102.336,E2 -7102.336} C_VEL
LIN {X 0,Y 474.333,Z 642.61,A -85,B 0,C 180,E1 -7104.047,E2 -7104.047} C_VEL
LIN {X 0,Y 474.355,Z 640.11,A -85,B 0,C 180,E1 -7105.752,E2 -7105.752} C_VEL
LIN {X 0,Y 474.608,Z 636.373,A -85,B 0,C 180,E1 -7107.454,E2 -7107.454} C_VEL
LIN {X 0,Y 474.801,Z 631.426,A -85,B 0,C 180,E1 -7109.152,E2 -7109.152} C_VEL
LIN {X 0,Y 475.203,Z 625.1,A -85,B 0,C 180,E1 -7110.848,E2 -7110.848} C_VEL
LIN {X 0,Y 475.683,Z 618.286,A -85,B 0,C 180,E1 -7112.329,E2 -7112.329} C_VEL
LIN {X 0,Y 476.211,Z 610.129,A -85,B 0,C 180,E1 -7113.808,E2 -7113.808} C_VEL
LIN {X 0,Y 476.942,Z 600.312,A -85,B 0,C 180,E1 -7115.284,E2 -7115.284} C_VEL
LIN {X 0,Y 477.583,Z 590.315,A -85,B 0,C 180,E1 -7116.549,E2 -7116.549} C_VEL
LIN {X 0,Y 478.254,Z 578.368,A -85,B 0,C 180,E1 -7117.813,E2 -7117.813} C_VEL
LIN {X 0,Y 479.028,Z 566.373,A -85,B 0,C 180,E1 -7118.862,E2 -7118.862} C_VEL
LIN {X 0,Y 479.765,Z 553.279,A -85,B 0,C 180,E1 -7119.805,E2 -7119.805} C_VEL
LIN {X 0,Y 480.341,Z 539.752,A -85,B 0,C 180,E1 -7120.592,E2 -7120.592} C_VEL
LIN {X 0,Y 480.876,Z 525.315,A -85,B 0,C 180,E1 -7121.242,E2 -7121.242} C_VEL
LIN {X 0,Y 481.13,Z 510.184,A -85,B 0,C 180,E1 -7121.747,E2 -7121.747} C_VEL
LIN {X 0,Y 481.272,Z 495.651,A -85,B 0,C 180,E1 -7122.064,E2 -7122.064} C_VEL
LIN {X 0,Y 482.312,Z 389.675,A -85,B 0,C 180,E1 -7123.687,E2 -7123.687} C_VEL
LIN {X 0,Y 474.746,Z 372.72,A -85,B 0,C 180,E1 -7124.334,E2 -7124.334} C_VEL
LIN {X 0,Y 474.609,Z 371.991,A -85,B 0,C 180,E1 -7124.362,E2 -7124.362} C_VEL
LIN {X 0,Y 474.595,Z 371.99,A -85,B 0,C 180,E1 -7127.227,E2 -7127.227} C_VEL
LIN {X 0,Y 474.616,Z 371.987,A -85,B 0,C 180,E1 -7129.912,E2 -7129.912} C_VEL
LIN {X 0,Y 474.576,Z 371.995,A -85,B 0,C 180,E1 -7132.646,E2 -7132.646} C_VEL
LIN {X 0,Y 474.595,Z 371.994,A -85,B 0,C 180,E1 -7135.432,E2 -7135.432} C_VEL
LIN {X 0,Y 474.588,Z 371.991,A -85,B 0,C 180,E1 -7138.286,E2 -7138.286} C_VEL
LIN {X 0,Y 474.573,Z 371.995,A -85,B 0,C 180,E1 -7141.219,E2 -7141.219} C_VEL
LIN {X 0,Y 474.605,Z 371.986,A -85,B 0,C 180,E1 -7144.243,E2 -7144.243} C_VEL
LIN {X 0,Y 474.536,Z 372.001,A -85,B 0,C 180,E1 -7147.388,E2 -7147.388} C_VEL
LIN {X 0,Y 474.578,Z 371.99,A -85,B 0,C 180,E1 -7149.64,E2 -7149.64} C_VEL
LIN {X 0,Y 474.571,Z 371.991,A -85,B 0,C 180,E1 -7152.229,E2 -7152.229} C_VEL
LIN {X 0,Y 474.606,Z 371.994,A -85,B 0,C 180,E1 -7155.298,E2 -7155.298} C_VEL
LIN {X 0,Y 474.587,Z 371.988,A -85,B 0,C 180,E1 -7158.211,E2 -7158.211} C_VEL
LIN {X 0,Y 474.611,Z 371.987,A -85,B 0,C 180,E1 -7160.45,E2 -7160.45} C_VEL
LIN {X 0,Y 474.572,Z 371.995,A -85,B 0,C 180,E1 -7163.675,E2 -7163.675} C_VEL
LIN {X 0,Y 474.601,Z 371.986,A -85,B 0,C 180,E1 -7166.776,E2 -7166.776} C_VEL
LIN {X 0,Y 474.543,Z 371.995,A -85,B 0,C 180,E1 -7169.765,E2 -7169.765} C_VEL
LIN {X 0,Y 474.594,Z 371.989,A -85,B 0,C 180,E1 -7172.684,E2 -7172.684} C_VEL
LIN {X 0,Y 474.611,Z 371.988,A -85,B 0,C 180,E1 -7175.504,E2 -7175.504} C_VEL
LIN {X 0,Y 474.626,Z 371.987,A -85,B 0,C 180,E1 -7178.884,E2 -7178.884} C_VEL
LIN {X 0,Y 474.632,Z 371.984,A -85,B 0,C 180,E1 -7181.883,E2 -7181.883} C_VEL
LIN {X 0,Y 474.688,Z 371.976,A -85,B 0,C 180,E1 -7184.544,E2 -7184.544} C_VEL
LIN {X 0,Y 474.694,Z 371.96,A -85,B 0,C 180,E1 -7188.037,E2 -7188.037} C_VEL
LIN {X 0,Y 474.651,Z 371.976,A -85,B 0,C 180,E1 -7191.485,E2 -7191.485} C_VEL
LIN {X 0,Y 474.726,Z 371.973,A -85,B 0,C 180,E1 -7194.052,E2 -7194.052} C_VEL
LIN {X 0,Y 474.833,Z 371.959,A -85,B 0,C 180,E1 -7197.455,E2 -7197.455} C_VEL
LIN {X 0,Y 474.865,Z 371.957,A -85,B 0,C 180,E1 -7200,E2 -7200} C_VEL
LIN {X 0,Y 474.867,Z 371.951,A -85,B 0,C 180,E1 -7202.545,E2 -7202.545} C_VEL
LIN {X 0,Y 474.716,Z 371.976,A -85,B 0,C 180,E1 -7205.948,E2 -7205.948} C_VEL
LIN {X 0,Y 474.655,Z 371.977,A -85,B 0,C 180,E1 -7208.515,E2 -7208.515} C_VEL
LIN {X 0,Y 474.694,Z 371.979,A -85,B 0,C 180,E1 -7211.962,E2 -7211.962} C_VEL
LIN {X 0,Y 474.642,Z 371.99,A -85,B 0,C 180,E1 -7215.755,E2 -7215.755} C_VEL
LIN {X 0,Y 474.593,Z 371.986,A -85,B 0,C 180,E1 -7219.013,E2 -7219.013} C_VEL
LIN {X 0,Y 474.565,Z 371.998,A -85,B 0,C 180,E1 -7221.73,E2 -7221.73} C_VEL
LIN {X 0,Y 474.615,Z 371.986,A -85,B 0,C 180,E1 -7224.495,E2 -7224.495} C_VEL
LIN {X 0,Y 474.588,Z 371.99,A -85,B 0,C 180,E1 -7227.327,E2 -7227.327} C_VEL
LIN {X 0,Y 474.585,Z 371.993,A -85,B 0,C 180,E1 -7230.231,E2 -7230.231} C_VEL
LIN {X 0,Y 474.605,Z 371.986,A -85,B 0,C 180,E1 -7233.223,E2 -7233.223} C_VEL
LIN {X 0,Y 474.562,Z 371.996,A -85,B 0,C 180,E1 -7236.326,E2 -7236.326} C_VEL
LIN {X 0,Y 474.591,Z 371.99,A -85,B 0,C 180,E1 -7239.644,E2 -7239.644} C_VEL
LIN {X 0,Y 474.568,Z 371.992,A -85,B 0,C 180,E1 -7242.23,E2 -7242.23} C_VEL
LIN {X 0,Y 474.609,Z 371.988,A -85,B 0,C 180,E1 -7245.298,E2 -7245.298} C_VEL
LIN {X 0,Y 474.579,Z 371.987,A -85,B 0,C 180,E1 -7248.211,E2 -7248.211} C_VEL
LIN {X 0,Y 474.581,Z 371.995,A -85,B 0,C 180,E1 -7251.54,E2 -7251.54} C_VEL
LIN {X 0,Y 474.637,Z 371.988,A -85,B 0,C 180,E1 -7255.245,E2 -7255.245} C_VEL
LIN {X 0,Y 474.671,Z 372.069,A -85,B 0,C 180,E1 -7255.602,E2 -7255.602} C_VEL
LIN {X 0,Y 480.515,Z 394.48,A -85,B 0,C 180,E1 -7258.577,E2 -7258.577} C_VEL
LIN {X 0,Y 480.547,Z 398.887,A -85,B 0,C 180,E1 -7259.09,E2 -7259.09} C_VEL
LIN {X 0,Y 479.594,Z 420.746,A -85,B 0,C 180,E1 -7261.551,E2 -7261.551} C_VEL
LIN {X 0,Y 478.564,Z 445.724,A -85,B 0,C 180,E1 -7264.328,E2 -7264.328} C_VEL
LIN {X 0,Y 477.902,Z 462.992,A -85,B 0,C 180,E1 -7266.232,E2 -7266.232} C_VEL
LIN {X 0,Y 482.07,Z 492.528,A -85,B 0,C 180,E1 -7266.901,E2 -7266.901} C_VEL
LIN {X 0,Y 480.555,Z 631.937,A -85,B 0,C 180,E1 -7269.032,E2 -7269.032} C_VEL
LIN {X 0,Y 480.043,Z 647.445,A -85,B 0,C 180,E1 -7269.429,E2 -7269.429} C_VEL
LIN {X 0,Y 479.321,Z 662.619,A -85,B 0,C 180,E1 -7269.991,E2 -7269.991} C_VEL
LIN {X 0,Y 478.554,Z 677.109,A -85,B 0,C 180,E1 -7270.705,E2 -7270.705} C_VEL
LIN {X 0,Y 477.812,Z 690.895,A -85,B 0,C 180,E1 -7271.565,E2 -7271.565} C_VEL
LIN {X 0,Y 476.961,Z 704.933,A -85,B 0,C 180,E1 -7272.64,E2 -7272.64} C_VEL
LIN {X 0,Y 476.196,Z 717.667,A -85,B 0,C 180,E1 -7273.825,E2 -7273.825} C_VEL
LIN {X 0,Y 475.434,Z 730.192,A -85,B 0,C 180,E1 -7275.227,E2 -7275.227} C_VEL
LIN {X 0,Y 474.889,Z 741.365,A -85,B 0,C 180,E1 -7276.739,E2 -7276.739} C_VEL
LIN {X 0,Y 474.446,Z 750.684,A -85,B 0,C 180,E1 -7278.248,E2 -7278.248} C_VEL
LIN {X 0,Y 474.243,Z 758.449,A -85,B 0,C 180,E1 -7279.756,E2 -7279.756} C_VEL
LIN {X 0,Y 474.082,Z 765.711,A -85,B 0,C 180,E1 -7281.475,E2 -7281.475} C_VEL
LIN {X 0,Y 474.022,Z 772.06,A -85,B 0,C 180,E1 -7283.394,E2 -7283.394} C_VEL
LIN {X 0,Y 474.006,Z 775.77,A -85,B 0,C 180,E1 -7284.896,E2 -7284.896} C_VEL
LIN {X 0,Y 474.067,Z 777.455,A -85,B 0,C 180,E1 -7285.749,E2 -7285.749} C_VEL
LIN {X 0,Y 473.997,Z 779.86,A -85,B 0,C 180,E1 -7287.45,E2 -7287.45} C_VEL
LIN {X 0,Y 474.038,Z 781.075,A -85,B 0,C 180,E1 -7289.15,E2 -7289.15} C_VEL
LIN {X 0,Y 474.038,Z 781.061,A -85,B 0,C 180,E1 -7290.849,E2 -7290.849} C_VEL
LIN {X 0,Y 474.002,Z 779.818,A -85,B 0,C 180,E1 -7292.549,E2 -7292.549} C_VEL
LIN {X 0,Y 474.067,Z 777.386,A -85,B 0,C 180,E1 -7294.25,E2 -7294.25} C_VEL
LIN {X 0,Y 474.016,Z 773.681,A -85,B 0,C 180,E1 -7295.957,E2 -7295.957} C_VEL
LIN {X 0,Y 474.042,Z 768.64,A -85,B 0,C 180,E1 -7297.667,E2 -7297.667} C_VEL
LIN {X 0,Y 474.133,Z 762.128,A -85,B 0,C 180,E1 -7299.383,E2 -7299.383} C_VEL
LIN {X 0,Y 474.379,Z 753.984,A -85,B 0,C 180,E1 -7301.104,E2 -7301.104} C_VEL
LIN {X 0,Y 474.711,Z 745.249,A -85,B 0,C 180,E1 -7302.628,E2 -7302.628} C_VEL
LIN {X 0,Y 475.194,Z 734.978,A -85,B 0,C 180,E1 -7304.124,E2 -7304.124} C_VEL
LIN {X 0,Y 475.763,Z 724.427,A -85,B 0,C 180,E1 -7305.42,E2 -7305.42} C_VEL
LIN {X 0,Y 476.499,Z 712.213,A -85,B 0,C 180,E1 -7306.683,E2 -7306.683} C_VEL
LIN {X 0,Y 477.253,Z 699.38,A -85,B 0,C 180,E1 -7307.791,E2 -7307.791} C_VEL
LIN {X 0,Y 477.995,Z 685.806,A -85,B 0,C 180,E1 -7308.761,E2 -7308.761} C_VEL
LIN {X 0,Y 478.873,Z 670.914,A -85,B 0,C 180,E1 -7309.615,E2 -7309.615} C_VEL
LIN {X 0,Y 479.663,Z 655.595,A -85,B 0,C 180,E1 -7310.294,E2 -7310.294} C_VEL
LIN {X 0,Y 480.311,Z 640.376,A -85,B 0,C 180,E1 -7310.782,E2 -7310.782} C_VEL
LIN {X 0,Y 480.701,Z 625.314,A -85,B 0,C 180,E1 -7311.101,E2 -7311.101} C_VEL
LIN {X 0,Y 482.193,Z 491.92,A -85,B 0,C 180,E1 -7313.141,E2 -7313.141} C_VEL
LIN {X 0,Y 477.929,Z 462.259,A -85,B 0,C 180,E1 -7313.852,E2 -7313.852} C_VEL
LIN {X 0,Y 479.249,Z 431.773,A -85,B 0,C 180,E1 -7317.274,E2 -7317.274} C_VEL
LIN {X 0,Y 480.605,Z 403.708,A -85,B 0,C 180,E1 -7320.492,E2 -7320.492} C_VEL
LIN {X 0,Y 480.901,Z 395.166,A -85,B 0,C 180,E1 -7321.496,E2 -7321.496} C_VEL
LIN {X 0,Y 476.855,Z 379.881,A -85,B 0,C 180,E1 -7323.623,E2 -7323.623} C_VEL
LIN {X 0,Y 474.63,Z 371.987,A -85,B 0,C 180,E1 -7324.786,E2 -7324.786} C_VEL
LIN {X 0,Y 474.581,Z 371.996,A -85,B 0,C 180,E1 -7328.459,E2 -7328.459} C_VEL
LIN {X 0,Y 474.592,Z 371.989,A -85,B 0,C 180,E1 -7330.954,E2 -7330.954} C_VEL
LIN {X 0,Y 474.592,Z 371.992,A -85,B 0,C 180,E1 -7334.105,E2 -7334.105} C_VEL
LIN {X 0,Y 474.555,Z 371.993,A -85,B 0,C 180,E1 -7337.059,E2 -7337.059} C_VEL
LIN {X 0,Y 474.58,Z 371.99,A -85,B 0,C 180,E1 -7339.339,E2 -7339.339} C_VEL
LIN {X 0,Y 474.578,Z 371.99,A -85,B 0,C 180,E1 -7341.707,E2 -7341.707} C_VEL
LIN {X 0,Y 474.597,Z 371.992,A -85,B 0,C 180,E1 -7344.724,E2 -7344.724} C_VEL
LIN {X 0,Y 474.607,Z 371.99,A -85,B 0,C 180,E1 -7347.786,E2 -7347.786} C_VEL
LIN {X 0,Y 474.584,Z 371.993,A -85,B 0,C 180,E1 -7350.89,E2 -7350.89} C_VEL
LIN {X 0,Y 474.575,Z 371.993,A -85,B 0,C 180,E1 -7353.623,E2 -7353.623} C_VEL
LIN {X 0,Y 474.583,Z 371.996,A -85,B 0,C 180,E1 -7356.652,E2 -7356.652} C_VEL
LIN {X 0,Y 474.596,Z 371.991,A -85,B 0,C 180,E1 -7360.087,E2 -7360.087} C_VEL
LIN {X 0,Y 474.573,Z 371.995,A -85,B 0,C 180,E1 -7362.772,E2 -7362.772} C_VEL
LIN {X 0,Y 474.611,Z 371.986,A -85,B 0,C 180,E1 -7365.42,E2 -7365.42} C_VEL
LIN {X 0,Y 474.688,Z 371.98,A -85,B 0,C 180,E1 -7368.037,E2 -7368.037} C_VEL
LIN {X 0,Y 474.651,Z 371.982,A -85,B 0,C 180,E1 -7371.485,E2 -7371.485} C_VEL
LIN {X 0,Y 474.712,Z 371.973,A -85,B 0,C 180,E1 -7374.052,E2 -7374.052} C_VEL
LIN {X 0,Y 474.864,Z 371.951,A -85,B 0,C 180,E1 -7377.455,E2 -7377.455} C_VEL
LIN {X 0,Y 474.801,Z 371.964,A -85,B 0,C 180,E1 -7380.848,E2 -7380.848} C_VEL
LIN {X 0,Y 474.862,Z 371.96,A -85,B 0,C 180,E1 -7382.545,E2 -7382.545} C_VEL
LIN {X 0,Y 474.742,Z 371.963,A -85,B 0,C 180,E1 -7385.948,E2 -7385.948} C_VEL
LIN {X 0,Y 474.686,Z 371.971,A -85,B 0,C 180,E1 -7388.514,E2 -7388.514} C_VEL
LIN {X 0,Y 474.689,Z 371.977,A -85,B 0,C 180,E1 -7391.963,E2 -7391.963} C_VEL
LIN {X 0,Y 474.667,Z 371.974,A -85,B 0,C 180,E1 -7395.768,E2 -7395.768} C_VEL
LIN {X 0,Y 474.65,Z 371.981,A -85,B 0,C 180,E1 -7399.011,E2 -7399.011} C_VEL
LIN {X 0,Y 474.575,Z 371.984,A -85,B 0,C 180,E1 -7401.73,E2 -7401.73} C_VEL
LIN {X 0,Y 474.613,Z 371.991,A -85,B 0,C 180,E1 -7404.496,E2 -7404.496} C_VEL
LIN {X 0,Y 474.588,Z 371.988,A -85,B 0,C 180,E1 -7407.327,E2 -7407.327} C_VEL
LIN {X 0,Y 474.589,Z 371.992,A -85,B 0,C 180,E1 -7410.232,E2 -7410.232} C_VEL
LIN {X 0,Y 474.604,Z 371.993,A -85,B 0,C 180,E1 -7413.223,E2 -7413.223} C_VEL
LIN {X 0,Y 474.579,Z 371.991,A -85,B 0,C 180,E1 -7416.325,E2 -7416.325} C_VEL
LIN {X 0,Y 474.613,Z 371.986,A -85,B 0,C 180,E1 -7419.549,E2 -7419.549} C_VEL
LIN {X 0,Y 474.576,Z 371.992,A -85,B 0,C 180,E1 -7422.232,E2 -7422.232} C_VEL
LIN {X 0,Y 474.609,Z 371.992,A -85,B 0,C 180,E1 -7425.299,E2 -7425.299} C_VEL
LIN {X 0,Y 474.597,Z 371.99,A -85,B 0,C 180,E1 -7428.214,E2 -7428.214} C_VEL
LIN {X 0,Y 474.603,Z 371.988,A -85,B 0,C 180,E1 -7431.543,E2 -7431.543} C_VEL
LIN {X 0,Y 474.615,Z 371.989,A -85,B 0,C 180,E1 -7434.726,E2 -7434.726} C_VEL
LIN {X 0,Y 474.624,Z 371.989,A -85,B 0,C 180,E1 -7437.531,E2 -7437.531} C_VEL
LIN {X 0,Y 475.674,Z 374.959,A -85,B 0,C 180,E1 -7437.653,E2 -7437.653} C_VEL
LIN {X 0,Y 482.685,Z 389.957,A -85,B 0,C 180,E1 -7438.3,E2 -7438.3} C_VEL
LIN {X 0,Y 481.746,Z 473.617,A -85,B 0,C 180,E1 -7439.594,E2 -7439.594} C_VEL
LIN {X 0,Y 481.093,Z 479.481,A -85,B 0,C 180,E1 -7439.648,E2 -7439.648} C_VEL
LIN {X 0,Y 475.651,Z 498.57,A -85,B 0,C 180,E1 -7439.665,E2 -7439.665} C_VEL
LIN {X 0,Y 475.018,Z 504.372,A -85,B 0,C 180,E1 -7439.763,E2 -7439.763} C_VEL
LIN {X 0,Y 474.697,Z 520.088,A -85,B 0,C 180,E1 -7440.206,E2 -7440.206} C_VEL
LIN {X 0,Y 474.32,Z 534.426,A -85,B 0,C 180,E1 -7440.788,E2 -7440.788} C_VEL
LIN {X 0,Y 473.615,Z 549.213,A -85,B 0,C 180,E1 -7441.576,E2 -7441.576} C_VEL
LIN {X 0,Y 472.953,Z 562.199,A -85,B 0,C 180,E1 -7442.452,E2 -7442.452} C_VEL
LIN {X 0,Y 472.225,Z 574.681,A -85,B 0,C 180,E1 -7443.483,E2 -7443.483} C_VEL
LIN {X 0,Y 471.401,Z 586.143,A -85,B 0,C 180,E1 -7444.621,E2 -7444.621} C_VEL
LIN {X 0,Y 470.591,Z 597.63,A -85,B 0,C 180,E1 -7445.99,E2 -7445.99} C_VEL
